C03637=1127.481,11.957,-50.735,179.626,6.543,149.306
C03638=1127.475,12.208,-50.749,179.627,6.548,149.306
C03639=1127.470,12.457,-50.763,179.628,6.553,149.307
C03640=1127.465,12.706,-50.777,179.629,6.558,149.308
C03641=1127.460,12.956,-50.790,179.630,6.562,149.309
C03642=1127.455,13.205,-50.804,179.630,6.567,149.309
C03643=1127.450,13.455,-50.818,179.632,6.572,149.310
C03644=1127.445,13.706,-50.832,179.632,6.576,149.311
C03645=1127.439,13.955,-50.846,179.633,6.581,149.312
C03646=1127.435,14.204,-50.860,179.634,6.585,149.312
C03647=1127.430,14.454,-50.874,179.635,6.590,149.313
C03648=1127.424,14.703,-50.887,179.636,6.594,149.314
C03649=1127.419,14.953,-50.901,179.637,6.600,149.315
C03650=1127.414,15.203,-50.916,179.638,6.604,149.315
C03651=1127.409,15.451,-50.929,179.639,6.609,149.316
C03652=1127.404,15.702,-50.942,179.640,6.613,149.317
C03653=1127.399,15.951,-50.957,179.640,6.618,149.318
C03654=1127.393,16.200,-50.971,179.642,6.622,149.318
C03655=1127.388,16.450,-50.985,179.643,6.627,149.319
C03656=1127.384,16.700,-50.999,179.644,6.632,149.320
C03657=1127.378,16.949,-51.013,179.645,6.636,149.321
C03658=1127.373,17.199,-51.027,179.646,6.640,149.321
C03659=1127.368,17.449,-51.040,179.646,6.645,149.322
C03660=1127.363,17.698,-51.054,179.647,6.649,149.323
C03661=1127.358,17.947,-51.069,179.649,6.655,149.323
C03662=1127.353,18.197,-51.083,179.650,6.659,149.324
C03663=1127.348,18.447,-51.097,179.651,6.664,149.325
C03664=1127.343,18.696,-51.111,179.652,6.668,149.326
C03665=1127.338,18.945,-51.125,179.652,6.673,149.326
C03666=1127.333,19.195,-51.140,179.653,6.677,149.327
C03667=1127.328,19.445,-51.154,179.654,6.681,149.328
C03668=1127.322,19.694,-51.168,179.656,6.686,149.328
C03669=1127.317,19.944,-51.182,179.657,6.691,149.329
C03670=1127.312,20.193,-51.196,179.658,6.695,149.330
C03671=1127.308,20.409,-51.208,179.658,6.699,149.331
C03672=1127.303,20.624,-51.220,179.659,6.703,149.331
C03673=1127.299,20.839,-51.233,179.661,6.707,149.332
C03674=1127.294,21.054,-51.245,179.661,6.711,149.332
C03675=1127.290,21.270,-51.257,179.662,6.715,149.333
C03676=1127.286,21.485,-51.270,179.662,6.719,149.334
C03677=1127.281,21.700,-51.281,179.664,6.723,149.334
C03678=1127.277,21.915,-51.294,179.664,6.726,149.335
C03679=1127.272,22.165,-51.309,179.665,6.730,149.335
C03680=1127.267,22.414,-51.323,179.667,6.736,149.336
C03681=1127.262,22.664,-51.337,179.668,6.740,149.337
C03682=1127.257,22.914,-51.351,179.669,6.745,149.337
C03683=1127.252,23.163,-51.366,179.670,6.749,149.338
C03684=1127.246,23.412,-51.380,179.671,6.753,149.339
C03685=1127.241,23.662,-51.394,179.672,6.758,149.339
C03686=1127.237,23.912,-51.408,179.673,6.762,149.340
C03687=1127.231,24.161,-51.424,179.674,6.767,149.341
C03688=1127.226,24.411,-51.438,179.675,6.771,149.342
C03689=1127.221,24.661,-51.452,179.676,6.776,149.342
C03690=1127.216,24.910,-51.466,179.677,6.780,149.343
C03691=1127.211,25.159,-51.480,179.678,6.785,149.344
C03692=1127.206,25.408,-51.495,179.679,6.789,149.344
C03693=1127.201,25.658,-51.510,179.680,6.793,149.345
C03694=1127.195,25.908,-51.525,179.682,6.798,149.345
C03695=1127.190,26.158,-51.539,179.683,6.802,149.346
C03696=1127.186,26.407,-51.554,179.684,6.806,149.347
C03697=1127.181,26.657,-51.568,179.684,6.811,149.348
C03698=1127.175,26.906,-51.582,179.685,6.815,149.348
C03699=1127.170,27.155,-51.596,179.686,6.820,149.349
C03700=1127.165,27.405,-51.612,179.688,6.825,149.350
C03701=1127.160,27.654,-51.626,179.689,6.829,149.350
C03702=1127.155,27.904,-51.640,179.690,6.833,149.351
C03703=1127.150,28.153,-51.655,179.691,6.838,149.352
C03704=1127.145,28.403,-51.670,179.692,6.842,149.352
C03705=1127.140,28.653,-51.685,179.693,6.846,149.353
C03706=1127.135,28.902,-51.700,179.694,6.851,149.353
C03707=1127.130,29.152,-51.714,179.695,6.855,149.354
C03708=1127.125,29.402,-51.728,179.696,6.859,149.355
C03709=1127.120,29.651,-51.744,179.697,6.863,149.355
C03710=1127.115,29.901,-51.758,179.699,6.868,149.356
C03711=1127.110,30.150,-51.773,179.700,6.872,149.357
C03712=1127.105,30.400,-51.788,179.701,6.876,149.357
C03713=1127.100,30.649,-51.802,179.702,6.881,149.358
C03714=1127.094,30.898,-51.817,179.703,6.886,149.359
C03715=1127.089,31.148,-51.832,179.704,6.890,149.359
C03716=1127.084,31.397,-51.847,179.706,6.894,149.360
C03717=1127.079,31.647,-51.861,179.707,6.898,149.360
C03718=1127.074,31.896,-51.876,179.708,6.903,149.361
C03719=1127.069,32.146,-51.891,179.709,6.907,149.362
C03720=1127.064,32.395,-51.906,179.710,6.911,149.362
C03721=1127.058,32.645,-51.921,179.711,6.916,149.363
C03722=1127.054,32.894,-51.936,179.712,6.920,149.364
C03723=1127.049,33.144,-51.950,179.713,6.924,149.364
C03724=1127.044,33.394,-51.966,179.714,6.929,149.365
C03725=1127.039,33.643,-51.981,179.716,6.933,149.366
C03726=1127.034,33.893,-51.995,179.717,6.937,149.366
C03727=1127.030,34.108,-52.008,179.718,6.941,149.367
C03728=1127.025,34.323,-52.021,179.719,6.944,149.367
C03729=1127.021,34.537,-52.034,179.720,6.949,149.368
C03730=1127.017,34.753,-52.047,179.721,6.952,149.368
C03731=1127.012,34.968,-52.060,179.722,6.956,149.369
C03732=1127.008,35.183,-52.073,179.723,6.959,149.369
C03733=1127.003,35.398,-52.085,179.724,6.963,149.370
C03734=1126.999,35.614,-52.099,179.725,6.967,149.370
C03735=1126.994,35.863,-52.114,179.726,6.971,149.371
C03736=1126.989,36.112,-52.129,179.727,6.975,149.372
C03737=1126.983,36.363,-52.144,179.728,6.980,149.372
C03738=1126.979,36.612,-52.159,179.730,6.983,149.373
C03739=1126.974,36.861,-52.174,179.731,6.988,149.373
C03740=1126.968,37.111,-52.189,179.732,6.992,149.374
C03741=1126.964,37.360,-52.204,179.733,6.996,149.375
C03742=1126.958,37.609,-52.219,179.734,7.001,149.375
C03743=1126.954,37.859,-52.235,179.736,7.005,149.376
C03744=1126.949,38.109,-52.250,179.737,7.009,149.376
C03745=1126.943,38.358,-52.265,179.738,7.013,149.377
C03746=1126.939,38.608,-52.280,179.739,7.018,149.378
C03747=1126.933,38.857,-52.296,179.740,7.021,149.378
C03748=1126.929,39.106,-52.311,179.741,7.026,149.379
C03749=1126.923,39.356,-52.326,179.742,7.030,149.379
C03750=1126.918,39.605,-52.341,179.744,7.034,149.380
C03751=1126.913,39.855,-52.357,179.745,7.038,149.380
C03752=1126.909,40.104,-52.372,179.746,7.043,149.381
C03753=1126.903,40.354,-52.387,179.747,7.047,149.382
C03754=1126.898,40.603,-52.403,179.748,7.051,149.382
C03755=1126.893,40.853,-52.417,179.750,7.055,149.383
C03756=1126.888,41.102,-52.433,179.751,7.059,149.383
C03757=1126.884,41.352,-52.448,179.752,7.064,149.384
C03758=1126.878,41.601,-52.464,179.753,7.068,149.384
C03759=1126.873,41.851,-52.479,179.755,7.072,149.385
C03760=1126.868,42.100,-52.494,179.756,7.076,149.386
C03761=1126.863,42.349,-52.510,179.757,7.080,149.386
C03762=1126.858,42.599,-52.526,179.758,7.085,149.387
C03763=1126.853,42.849,-52.541,179.759,7.089,149.387
C03764=1126.848,43.098,-52.556,179.761,7.093,149.388
C03765=1126.843,43.347,-52.572,179.762,7.097,149.389
C03766=1126.838,43.596,-52.587,179.763,7.101,149.389
C03767=1126.833,43.847,-52.603,179.765,7.105,149.390
C03768=1126.828,44.096,-52.618,179.766,7.110,149.390
C03769=1126.823,44.345,-52.633,179.767,7.114,149.391
C03770=1126.818,44.594,-52.649,179.768,7.118,149.391
C03771=1126.813,44.845,-52.665,179.769,7.122,149.392
C03772=1126.808,45.094,-52.681,179.770,7.126,149.393
C03773=1126.803,45.343,-52.696,179.772,7.130,149.393
C03774=1126.798,45.593,-52.711,179.773,7.135,149.394
C03775=1126.793,45.843,-52.727,179.775,7.139,149.394
C03776=1126.787,46.092,-52.743,179.776,7.143,149.395
C03777=1126.783,46.341,-52.758,179.777,7.147,149.395
C03778=1126.778,46.591,-52.774,179.778,7.151,149.396
C03779=1126.773,46.840,-52.790,179.779,7.155,149.396
C03780=1126.767,47.089,-52.805,179.781,7.159,149.397
C03781=1126.763,47.339,-52.821,179.782,7.164,149.398
C03782=1126.758,47.588,-52.836,179.783,7.168,149.398
C03783=1126.753,47.803,-52.849,179.785,7.172,149.399
C03784=1126.750,48.018,-52.864,179.786,7.175,149.399
C03785=1126.744,48.234,-52.877,179.787,7.179,149.399
C03786=1126.741,48.449,-52.891,179.788,7.182,149.400
C03787=1126.736,48.664,-52.904,179.789,7.186,149.401
C03788=1126.732,48.879,-52.918,179.790,7.189,149.401
C03789=1126.728,49.094,-52.931,179.791,7.193,149.401
C03790=1126.724,49.309,-52.945,179.793,7.197,149.402
C03791=1126.719,49.558,-52.961,179.794,7.201,149.402
C03792=1126.713,49.808,-52.976,179.795,7.205,149.403
C03793=1126.709,50.058,-52.992,179.796,7.209,149.404
C03794=1126.703,50.306,-53.009,179.798,7.213,149.404
C03795=1126.698,50.556,-53.024,179.799,7.217,149.405
C03796=1126.693,50.806,-53.040,179.801,7.221,149.405
C03797=1126.688,51.055,-53.057,179.802,7.225,149.406
C03798=1126.684,51.305,-53.072,179.803,7.229,149.406
C03799=1126.679,51.554,-53.088,179.804,7.234,149.407
C03800=1126.674,51.803,-53.104,179.806,7.238,149.407
C03801=1126.669,52.053,-53.120,179.807,7.242,149.408
C03802=1126.664,52.302,-53.135,179.808,7.246,149.408
C03803=1126.659,52.552,-53.152,179.810,7.250,149.409
C03804=1126.654,52.801,-53.168,179.811,7.254,149.409
C03805=1126.648,53.051,-53.183,179.812,7.258,149.410
C03806=1126.644,53.300,-53.200,179.813,7.261,149.410
C03807=1126.638,53.549,-53.215,179.814,7.266,149.411
C03808=1126.634,53.799,-53.232,179.816,7.270,149.411
C03809=1126.629,54.048,-53.248,179.817,7.274,149.412
C03810=1126.624,54.298,-53.264,179.818,7.278,149.413
C03811=1126.619,54.547,-53.280,179.820,7.282,149.413
C03812=1126.614,54.796,-53.296,179.821,7.286,149.414
C03813=1126.609,55.046,-53.312,179.822,7.290,149.414
C03814=1126.604,55.295,-53.329,179.824,7.294,149.415
C03815=1126.599,55.545,-53.345,179.825,7.298,149.415
C03816=1126.594,55.794,-53.361,179.826,7.303,149.416
C03817=1126.589,56.044,-53.377,179.828,7.306,149.416
C03818=1126.584,56.293,-53.393,179.829,7.311,149.417
C03819=1126.579,56.543,-53.409,179.831,7.315,149.417
C03820=1126.574,56.792,-53.425,179.832,7.319,149.418
C03821=1126.569,57.042,-53.442,179.833,7.323,149.418
C03822=1126.564,57.291,-53.458,179.835,7.327,149.419
C03823=1126.559,57.541,-53.474,179.836,7.331,149.419
C03824=1126.554,57.790,-53.490,179.837,7.335,149.420
C03825=1126.549,58.039,-53.507,179.839,7.339,149.420
C03826=1126.544,58.288,-53.523,179.840,7.343,149.421
C03827=1126.539,58.538,-53.539,179.841,7.347,149.422
C03828=1126.534,58.787,-53.556,179.843,7.351,149.422
C03829=1126.529,59.037,-53.572,179.844,7.355,149.422
C03830=1126.524,59.286,-53.589,179.845,7.360,149.423
C03831=1126.519,59.535,-53.605,179.847,7.363,149.423
C03832=1126.514,59.785,-53.621,179.849,7.367,149.424
C03833=1126.509,60.034,-53.637,179.850,7.372,149.425
C03834=1126.505,60.284,-53.654,179.851,7.376,149.425
C03835=1126.499,60.534,-53.670,179.852,7.379,149.426
C03836=1126.494,60.783,-53.687,179.853,7.383,149.426
C03837=1126.489,61.032,-53.703,179.855,7.387,149.426
C03838=1126.485,61.281,-53.720,179.856,7.391,149.427
C03839=1126.480,61.497,-53.735,179.858,7.395,149.428
C03840=1126.476,61.711,-53.748,179.858,7.398,149.428
C03841=1126.471,61.926,-53.763,179.860,7.402,149.428
C03842=1126.468,62.141,-53.777,179.861,7.405,149.429
C03843=1126.463,62.356,-53.791,179.862,7.408,149.429
C03844=1126.459,62.571,-53.805,179.863,7.412,149.430
C03845=1126.455,62.786,-53.820,179.864,7.415,149.430
C03846=1126.450,63.001,-53.834,179.866,7.419,149.431
C03847=1126.446,63.251,-53.850,179.868,7.423,149.431
C03848=1126.440,63.500,-53.867,179.869,7.428,149.432
C03849=1126.435,63.749,-53.883,179.870,7.431,149.432
C03850=1126.431,63.999,-53.900,179.872,7.435,149.432
C03851=1126.425,64.248,-53.917,179.872,7.439,149.433
C03852=1126.420,64.497,-53.934,179.874,7.443,149.434
C03853=1126.416,64.747,-53.950,179.875,7.447,149.434
C03854=1126.411,64.996,-53.967,179.877,7.451,149.435
C03855=1126.406,65.246,-53.984,179.878,7.455,149.435
C03856=1126.401,65.495,-54.000,179.880,7.459,149.435
C03857=1126.396,65.744,-54.016,179.881,7.463,149.436
C03858=1126.391,65.994,-54.033,179.882,7.467,149.437
C03859=1126.386,66.244,-54.050,179.884,7.471,149.437
C03860=1126.381,66.492,-54.066,179.885,7.475,149.438
C03861=1126.376,66.742,-54.084,179.887,7.479,149.438
C03862=1126.371,66.992,-54.100,179.888,7.483,149.438
C03863=1126.366,67.242,-54.117,179.890,7.487,149.439
C03864=1126.361,67.490,-54.134,179.891,7.491,149.440
C03865=1126.357,67.740,-54.150,179.892,7.495,149.440
C03866=1126.352,67.989,-54.168,179.894,7.499,149.440
C03867=1126.347,68.238,-54.185,179.895,7.503,149.441
C03868=1126.341,68.488,-54.202,179.897,7.507,149.441
C03869=1126.337,68.737,-54.219,179.898,7.511,149.442
C03870=1126.332,68.987,-54.235,179.900,7.515,149.442
C03871=1126.327,69.236,-54.252,179.901,7.519,149.443
C03872=1126.322,69.485,-54.269,179.903,7.523,149.443
C03873=1126.317,69.735,-54.286,179.904,7.527,149.444
C03874=1126.312,69.984,-54.303,179.905,7.531,149.444
C03875=1126.307,70.233,-54.320,179.907,7.535,149.445
C03876=1126.302,70.482,-54.337,179.908,7.538,149.445
C03877=1126.297,70.732,-54.354,179.909,7.542,149.446
C03878=1126.293,70.982,-54.371,179.910,7.547,149.446
C03879=1126.287,71.231,-54.388,179.912,7.551,149.447
C03880=1126.282,71.480,-54.405,179.914,7.554,149.447
C03881=1126.277,71.729,-54.423,179.915,7.558,149.448
C03882=1126.273,71.979,-54.439,179.916,7.563,149.448
C03883=1126.268,72.229,-54.457,179.918,7.567,149.449
C03884=1126.263,72.477,-54.473,179.919,7.570,149.449
C03885=1126.258,72.727,-54.491,179.921,7.574,149.450
C03886=1126.253,72.976,-54.508,179.922,7.579,149.450
C03887=1126.248,73.226,-54.525,179.924,7.583,149.451
C03888=1126.243,73.476,-54.542,179.925,7.586,149.451
C03889=1126.239,73.725,-54.559,179.926,7.591,149.452
C03890=1126.233,73.974,-54.576,179.928,7.595,149.452
C03891=1126.228,74.223,-54.594,179.930,7.599,149.453
C03892=1126.224,74.472,-54.611,179.931,7.602,149.453
C03893=1126.218,74.722,-54.628,179.933,7.606,149.453
C03894=1126.214,74.972,-54.645,179.934,7.611,149.454
C03895=1126.210,75.186,-54.660,179.935,7.614,149.455
C03896=1126.205,75.402,-54.675,179.936,7.618,149.455
C03897=1126.201,75.616,-54.690,179.937,7.621,149.455
C03898=1126.196,75.831,-54.705,179.939,7.624,149.456
C03899=1126.192,76.046,-54.720,179.940,7.627,149.456
C03900=1126.189,76.260,-54.735,179.941,7.630,149.456
C03901=1126.184,76.476,-54.749,179.943,7.634,149.457
C03902=1126.180,76.690,-54.765,179.944,7.637,149.457
C03903=1126.175,76.940,-54.782,179.945,7.642,149.458
C03904=1126.171,77.189,-54.800,179.946,7.645,149.458
C03905=1126.165,77.438,-54.816,179.947,7.649,149.459
C03906=1126.160,77.687,-54.834,179.948,7.652,149.459
C03907=1126.155,77.937,-54.852,179.948,7.656,149.460
C03908=1126.150,78.186,-54.868,179.950,7.660,149.461
C03909=1126.145,78.436,-54.886,179.951,7.663,149.461
C03910=1126.140,78.685,-54.904,179.952,7.667,149.462
C03911=1126.136,78.934,-54.921,179.953,7.671,149.462
C03912=1126.131,79.183,-54.939,179.954,7.675,149.463
C03913=1126.126,79.433,-54.956,179.955,7.678,149.463
C03914=1126.121,79.682,-54.974,179.956,7.682,149.464
C03915=1126.116,79.932,-54.991,179.957,7.685,149.464
C03916=1126.111,80.181,-55.009,179.958,7.690,149.465
C03917=1126.106,80.431,-55.026,179.960,7.694,149.465
C03918=1126.101,80.680,-55.044,179.960,7.697,149.466
C03919=1126.096,80.929,-55.062,179.962,7.701,149.466
C03920=1126.091,81.178,-55.078,179.962,7.704,149.467
C03921=1126.086,81.427,-55.096,179.964,7.708,149.468
C03922=1126.081,81.677,-55.114,179.965,7.713,149.468
C03923=1126.076,81.926,-55.132,179.966,7.716,149.469
C03924=1126.071,82.175,-55.150,179.967,7.720,149.469
C03925=1126.067,82.425,-55.166,179.968,7.723,149.470
C03926=1126.062,82.674,-55.184,179.969,7.727,149.470
C03927=1126.057,82.923,-55.202,179.971,7.731,149.471
C03928=1126.052,83.173,-55.219,179.972,7.734,149.471
C03929=1126.047,83.422,-55.237,179.973,7.739,149.472
C03930=1126.042,83.671,-55.255,179.974,7.743,149.472
C03931=1126.037,83.921,-55.273,179.975,7.746,149.473
C03932=1126.033,84.170,-55.290,179.976,7.750,149.473
C03933=1126.028,84.419,-55.308,179.978,7.754,149.474
C03934=1126.023,84.669,-55.326,179.979,7.758,149.474
C03935=1126.018,84.919,-55.344,179.980,7.761,149.475
C03936=1126.013,85.168,-55.362,179.982,7.765,149.475
C03937=1126.008,85.417,-55.380,179.983,7.770,149.476
C03938=1126.003,85.666,-55.398,179.984,7.773,149.476
C03939=1125.998,85.916,-55.415,179.985,7.777,149.477
C03940=1125.993,86.165,-55.433,179.987,7.781,149.477
C03941=1125.988,86.415,-55.451,179.988,7.785,149.478
C03942=1125.983,86.664,-55.469,179.990,7.789,149.478
C03943=1125.979,86.913,-55.486,179.991,7.793,149.479
C03944=1125.974,87.162,-55.504,179.992,7.796,149.479
C03945=1125.969,87.412,-55.521,179.993,7.800,149.480
C03946=1125.964,87.661,-55.539,179.995,7.804,149.480
C03947=1125.959,87.910,-55.557,179.996,7.808,149.481
C03948=1125.954,88.159,-55.575,179.998,7.812,149.481
C03949=1125.950,88.409,-55.594,179.999,7.816,149.482
C03950=1125.945,88.658,-55.612,-179.999,7.820,149.482
C03951=1125.941,88.873,-55.627,-179.998,7.823,149.483
C03952=1125.936,89.088,-55.643,-179.997,7.826,149.483
C03953=1125.932,89.303,-55.658,-179.996,7.830,149.483
C03954=1125.928,89.517,-55.674,-179.995,7.833,149.484
C03955=1125.924,89.732,-55.689,-179.994,7.836,149.484
C03956=1125.920,89.947,-55.705,-179.992,7.840,149.485
C03957=1125.916,90.162,-55.720,-179.991,7.843,149.485
C03958=1125.911,90.377,-55.736,-179.990,7.846,149.485
C03959=1125.906,90.626,-55.754,-179.988,7.850,149.486
C03960=1125.901,90.875,-55.772,-179.986,7.854,149.486
C03961=1125.896,91.124,-55.790,-179.985,7.858,149.487
C03962=1125.892,91.374,-55.808,-179.984,7.862,149.487
C03963=1125.887,91.623,-55.826,-179.982,7.866,149.488
C03964=1125.882,91.872,-55.844,-179.980,7.870,149.488
C03965=1125.877,92.121,-55.862,-179.979,7.873,149.489
C03966=1125.872,92.370,-55.881,-179.977,7.877,149.489
C03967=1125.867,92.619,-55.899,-179.976,7.881,149.489
C03968=1125.862,92.869,-55.918,-179.974,7.885,149.490
C03969=1125.857,93.119,-55.936,-179.973,7.889,149.490
C03970=1125.853,93.368,-55.954,-179.971,7.893,149.491
C03971=1125.848,93.617,-55.972,-179.969,7.898,149.491
C03972=1125.843,93.866,-55.990,-179.967,7.901,149.492
C03973=1125.838,94.116,-56.008,-179.965,7.905,149.492
C03974=1125.834,94.365,-56.027,-179.964,7.909,149.492
C03975=1125.828,94.614,-56.045,-179.962,7.913,149.493
C03976=1125.823,94.863,-56.063,-179.961,7.917,149.493
C03977=1125.819,95.113,-56.082,-179.959,7.921,149.493
C03978=1125.814,95.362,-56.100,-179.957,7.924,149.494
C03979=1125.809,95.611,-56.119,-179.955,7.928,149.494
C03980=1125.804,95.860,-56.137,-179.954,7.932,149.495
C03981=1125.799,96.110,-56.155,-179.952,7.936,149.495
C03982=1125.795,96.359,-56.173,-179.950,7.941,149.496
C03983=1125.790,96.608,-56.192,-179.948,7.945,149.496
C03984=1125.784,96.857,-56.211,-179.946,7.948,149.496
C03985=1125.780,97.107,-56.229,-179.945,7.952,149.497
C03986=1125.775,97.356,-56.248,-179.943,7.956,149.497
C03987=1125.770,97.605,-56.266,-179.942,7.960,149.498
C03988=1125.765,97.855,-56.284,-179.939,7.964,149.498
C03989=1125.761,98.104,-56.303,-179.937,7.968,149.498
C03990=1125.756,98.353,-56.321,-179.936,7.972,149.499
C03991=1125.751,98.603,-56.340,-179.934,7.976,149.499
C03992=1125.746,98.852,-56.359,-179.931,7.980,149.499
C03993=1125.741,99.101,-56.377,-179.930,7.984,149.500
C03994=1125.736,99.350,-56.395,-179.928,7.988,149.500
C03995=1125.732,99.600,-56.414,-179.926,7.991,149.500
C03996=1125.727,99.849,-56.432,-179.925,7.995,149.501
C03997=1125.722,100.098,-56.452,-179.922,8.000,149.501
C03998=1125.717,100.347,-56.470,-179.920,8.003,149.501
C03999=1125.712,100.596,-56.489,-179.919,8.007,149.502
C04000=1125.707,100.846,-56.508,-179.916,8.012,149.502
C04001=1125.703,101.095,-56.526,-179.914,8.015,149.502
C04002=1125.697,101.344,-56.545,-179.912,8.019,149.503
C04003=1125.693,101.594,-56.564,-179.911,8.023,149.503
C04004=1125.688,101.843,-56.583,-179.908,8.027,149.503
C04005=1125.683,102.092,-56.601,-179.906,8.031,149.504
C04006=1125.678,102.342,-56.620,-179.904,8.034,149.504
C04007=1125.674,102.556,-56.636,-179.903,8.038,149.504
C04008=1125.670,102.770,-56.653,-179.901,8.042,149.505
C04009=1125.666,102.986,-56.669,-179.899,8.045,149.505
C04010=1125.661,103.200,-56.685,-179.897,8.048,149.505
C04011=1125.657,103.415,-56.701,-179.896,8.052,149.506
C04012=1125.653,103.629,-56.718,-179.894,8.055,149.506
C04013=1125.650,103.844,-56.734,-179.891,8.059,149.506
C04014=1125.645,104.059,-56.750,-179.890,8.062,149.506
C04015=1125.640,104.308,-56.769,-179.888,8.066,149.507
C04016=1125.635,104.557,-56.788,-179.886,8.070,149.507
C04017=1125.630,104.806,-56.806,-179.883,8.074,149.507
C04018=1125.626,105.056,-56.826,-179.881,8.078,149.507
C04019=1125.621,105.305,-56.845,-179.879,8.082,149.508
C04020=1125.616,105.554,-56.864,-179.877,8.086,149.508
C04021=1125.611,105.804,-56.883,-179.875,8.089,149.508
C04022=1125.607,106.053,-56.902,-179.872,8.094,149.508
C04023=1125.601,106.302,-56.921,-179.870,8.098,149.509
C04024=1125.597,106.551,-56.940,-179.868,8.102,149.509
C04025=1125.592,106.800,-56.959,-179.866,8.105,149.509
C04026=1125.587,107.050,-56.979,-179.863,8.110,149.509
C04027=1125.582,107.299,-56.997,-179.861,8.113,149.510
C04028=1125.578,107.548,-57.017,-179.859,8.117,149.510
C04029=1125.573,107.797,-57.036,-179.857,8.121,149.510
C04030=1125.568,108.046,-57.055,-179.855,8.125,149.511
C04031=1125.563,108.295,-57.075,-179.852,8.129,149.511
C04032=1125.559,108.545,-57.093,-179.850,8.133,149.511
C04033=1125.553,108.794,-57.112,-179.847,8.137,149.511
C04034=1125.548,109.043,-57.132,-179.845,8.140,149.511
C04035=1125.544,109.293,-57.151,-179.842,8.145,149.512
C04036=1125.539,109.542,-57.170,-179.840,8.148,149.512
C04037=1125.534,109.791,-57.190,-179.838,8.152,149.512
C04038=1125.529,110.040,-57.209,-179.835,8.157,149.512
C04039=1125.525,110.289,-57.228,-179.833,8.160,149.513
C04040=1125.520,110.538,-57.247,-179.830,8.164,149.513
C04041=1125.515,110.788,-57.267,-179.828,8.168,149.513
C04042=1125.510,111.037,-57.287,-179.826,8.171,149.513
C04043=1125.506,111.286,-57.305,-179.824,8.175,149.513
C04044=1125.501,111.535,-57.325,-179.822,8.178,149.514
C04045=1125.496,111.784,-57.344,-179.820,8.182,149.514
C04046=1125.491,112.034,-57.364,-179.818,8.185,149.514
C04047=1125.486,112.283,-57.384,-179.816,8.189,149.514
C04048=1125.482,112.531,-57.403,-179.814,8.193,149.515
C04049=1125.477,112.781,-57.423,-179.812,8.196,149.515
C04050=1125.472,113.030,-57.442,-179.810,8.200,149.515
C04051=1125.467,113.279,-57.462,-179.808,8.204,149.516
C04052=1125.462,113.529,-57.481,-179.806,8.207,149.516
C04053=1125.457,113.779,-57.501,-179.804,8.211,149.516
C04054=1125.453,114.027,-57.520,-179.802,8.214,149.516
C04055=1125.448,114.276,-57.540,-179.801,8.217,149.516
C04056=1125.444,114.526,-57.560,-179.799,8.221,149.517
C04057=1125.438,114.774,-57.579,-179.797,8.224,149.517
C04058=1125.434,115.024,-57.599,-179.795,8.228,149.517
C04059=1125.429,115.274,-57.618,-179.793,8.231,149.518
C04060=1125.424,115.522,-57.638,-179.791,8.235,149.518
C04061=1125.419,115.771,-57.658,-179.789,8.239,149.518
C04062=1125.414,116.021,-57.678,-179.787,8.242,149.518
C04063=1125.410,116.235,-57.694,-179.786,8.245,149.519
C04064=1125.407,116.450,-57.712,-179.784,8.248,149.519
C04065=1125.402,116.664,-57.728,-179.782,8.251,149.519
C04066=1125.398,116.879,-57.745,-179.781,8.254,149.519
C04067=1125.394,117.094,-57.762,-179.779,8.257,149.520
C04068=1125.390,117.308,-57.780,-179.778,8.259,149.520
C04069=1125.385,117.522,-57.796,-179.776,8.263,149.520
C04070=1125.382,117.738,-57.814,-179.774,8.265,149.520
C04071=1125.377,117.986,-57.834,-179.772,8.269,149.520
C04072=1125.372,118.235,-57.853,-179.771,8.273,149.521
C04073=1125.367,118.485,-57.873,-179.769,8.276,149.521
C04074=1125.363,118.734,-57.893,-179.767,8.279,149.521
C04075=1125.358,118.983,-57.913,-179.765,8.283,149.522
C04076=1125.353,119.232,-57.933,-179.763,8.286,149.522
C04077=1125.348,119.481,-57.953,-179.762,8.290,149.522
C04078=1125.343,119.731,-57.972,-179.760,8.293,149.522
C04079=1125.339,119.980,-57.993,-179.758,8.296,149.523
C04080=1125.334,120.229,-58.012,-179.756,8.300,149.523
C04081=1125.329,120.478,-58.032,-179.754,8.303,149.523
C04082=1125.324,120.727,-58.052,-179.752,8.307,149.524
C04083=1125.320,120.976,-58.072,-179.751,8.310,149.524
C04084=1125.315,121.226,-58.092,-179.749,8.313,149.524
C04085=1125.310,121.475,-58.113,-179.747,8.317,149.524
C04086=1125.305,121.724,-58.132,-179.745,8.320,149.524
C04087=1125.300,121.973,-58.153,-179.744,8.323,149.525
C04088=1125.295,122.222,-58.172,-179.742,8.327,149.525
C04089=1125.291,122.471,-58.193,-179.740,8.330,149.525
C04090=1125.286,122.721,-58.212,-179.737,8.334,149.526
C04091=1125.282,122.970,-58.233,-179.736,8.337,149.526
C04092=1125.277,123.218,-58.253,-179.734,8.340,149.526
C04093=1125.272,123.468,-58.272,-179.732,8.344,149.526
C04094=1125.267,123.717,-58.293,-179.730,8.347,149.527
C04095=1125.262,123.966,-58.314,-179.729,8.350,149.527
C04096=1125.258,124.215,-58.333,-179.727,8.354,149.527
C04097=1125.253,124.464,-58.354,-179.725,8.357,149.527
C04098=1125.249,124.714,-58.373,-179.724,8.360,149.528
C04099=1125.243,124.963,-58.394,-179.722,8.364,149.528
C04100=1125.238,125.211,-58.414,-179.720,8.367,149.528
C04101=1125.234,125.460,-58.435,-179.718,8.371,149.529
C04102=1125.229,125.710,-58.454,-179.716,8.374,149.529
C04103=1125.225,125.959,-58.475,-179.714,8.377,149.529
C04104=1125.220,126.208,-58.496,-179.712,8.381,149.529
C04105=1125.215,126.458,-58.515,-179.711,8.384,149.530
C04106=1125.210,126.707,-58.536,-179.709,8.387,149.530
C04107=1125.206,126.956,-58.556,-179.707,8.391,149.530
C04108=1125.201,127.205,-58.577,-179.706,8.394,149.530
C04109=1125.196,127.454,-58.597,-179.704,8.397,149.531
C04110=1125.192,127.703,-58.617,-179.702,8.401,149.531
C04111=1125.187,127.952,-58.637,-179.701,8.404,149.531
C04112=1125.182,128.202,-58.658,-179.699,8.407,149.531
C04113=1125.178,128.451,-58.679,-179.697,8.411,149.532
C04114=1125.173,128.699,-58.699,-179.695,8.414,149.532
C04115=1125.167,128.949,-58.719,-179.693,8.417,149.532
C04116=1125.163,129.198,-58.739,-179.691,8.421,149.533
C04117=1125.158,129.447,-58.760,-179.690,8.424,149.533
C04118=1125.153,129.696,-58.781,-179.688,8.427,149.533
C04119=1125.149,129.910,-58.798,-179.687,8.430,149.533
C04120=1125.146,130.125,-58.816,-179.685,8.433,149.534
C04121=1125.141,130.339,-58.833,-179.684,8.435,149.534
C04122=1125.137,130.554,-58.851,-179.682,8.438,149.534
C04123=1125.133,130.769,-58.869,-179.681,8.441,149.535
C04124=1125.129,130.982,-58.887,-179.679,8.445,149.535
C04125=1125.125,131.197,-58.904,-179.678,8.447,149.535
C04126=1125.120,131.412,-58.922,-179.677,8.450,149.535
C04127=1125.116,131.661,-58.942,-179.675,8.453,149.535
C04128=1125.112,131.910,-58.963,-179.673,8.457,149.536
C04129=1125.106,132.159,-58.984,-179.671,8.460,149.536
C04130=1125.102,132.408,-59.004,-179.670,8.463,149.536
C04131=1125.097,132.658,-59.025,-179.668,8.466,149.537
C04132=1125.092,132.907,-59.045,-179.667,8.470,149.537
C04133=1125.087,133.156,-59.066,-179.665,8.473,149.537
C04134=1125.083,133.405,-59.087,-179.663,8.477,149.537
C04135=1125.078,133.653,-59.108,-179.662,8.480,149.538
C04136=1125.073,133.902,-59.129,-179.660,8.483,149.538
C04137=1125.069,134.151,-59.149,-179.659,8.486,149.539
C04138=1125.064,134.401,-59.170,-179.657,8.490,149.539
C04139=1125.059,134.650,-59.190,-179.654,8.493,149.539
C04140=1125.054,134.899,-59.211,-179.653,8.496,149.539
C04141=1125.050,135.148,-59.232,-179.651,8.500,149.540
C04142=1125.045,135.398,-59.253,-179.650,8.503,149.540
C04143=1125.041,135.647,-59.274,-179.648,8.506,149.540
C04144=1125.036,135.896,-59.294,-179.647,8.509,149.541
C04145=1125.031,136.144,-59.316,-179.645,8.513,149.541
C04146=1125.026,136.393,-59.337,-179.643,8.516,149.541
C04147=1125.021,136.643,-59.358,-179.642,8.519,149.541
C04148=1125.017,136.892,-59.378,-179.640,8.523,149.542
C04149=1125.011,137.141,-59.399,-179.639,8.526,149.542
C04150=1125.008,137.390,-59.420,-179.637,8.530,149.543
C04151=1125.003,137.639,-59.441,-179.636,8.532,149.543
C04152=1124.998,137.888,-59.462,-179.633,8.536,149.543
C04153=1124.993,138.137,-59.483,-179.632,8.539,149.543
C04154=1124.988,138.387,-59.504,-179.630,8.542,149.544
C04155=1124.984,138.635,-59.525,-179.629,8.546,149.544
C04156=1124.979,138.884,-59.546,-179.627,8.549,149.544
C04157=1124.975,139.134,-59.566,-179.626,8.553,149.545
C04158=1124.970,139.383,-59.588,-179.624,8.556,149.545
C04159=1124.965,139.632,-59.609,-179.623,8.559,149.545
C04160=1124.960,139.881,-59.629,-179.621,8.562,149.546
C04161=1124.955,140.130,-59.650,-179.620,8.566,149.546
C04162=1124.951,140.378,-59.671,-179.618,8.569,149.546
C04163=1124.946,140.628,-59.693,-179.616,8.573,149.547
C04164=1124.942,140.877,-59.714,-179.615,8.575,149.547
C04165=1124.937,141.126,-59.735,-179.613,8.579,149.547
C04166=1124.932,141.375,-59.756,-179.612,8.582,149.548
C04167=1124.927,141.624,-59.777,-179.610,8.586,149.548
C04168=1124.923,141.874,-59.798,-179.609,8.588,149.548
C04169=1124.918,142.123,-59.819,-179.607,8.592,149.549
C04170=1124.913,142.371,-59.841,-179.606,8.595,149.549
C04171=1124.909,142.620,-59.861,-179.604,8.599,149.549
C04172=1124.904,142.869,-59.883,-179.603,8.602,149.550
C04173=1124.899,143.119,-59.904,-179.601,8.606,149.550
C04174=1124.895,143.368,-59.926,-179.600,8.609,149.550
C04175=1124.891,143.582,-59.944,-179.599,8.611,149.551
C04176=1124.886,143.797,-59.962,-179.598,8.614,149.551
C04177=1124.883,144.011,-59.981,-179.596,8.617,149.551
C04178=1124.878,144.225,-59.999,-179.595,8.620,149.552
C04179=1124.874,144.439,-60.016,-179.594,8.623,149.552
C04180=1124.870,144.654,-60.035,-179.592,8.626,149.552
C04181=1124.866,144.868,-60.054,-179.591,8.629,149.553
C04182=1124.862,145.083,-60.072,-179.590,8.631,149.553
C04183=1124.857,145.332,-60.093,-179.587,8.636,149.553
C04184=1124.852,145.581,-60.114,-179.584,8.640,149.553
C04185=1124.848,145.830,-60.136,-179.582,8.643,149.554
C04186=1124.844,146.078,-60.157,-179.579,8.647,149.554
C04187=1124.839,146.328,-60.178,-179.576,8.652,149.554
C04188=1124.834,146.577,-60.200,-179.574,8.655,149.554
C04189=1124.829,146.826,-60.221,-179.572,8.659,149.554
C04190=1124.824,147.075,-60.243,-179.569,8.663,149.555
C04191=1124.820,147.324,-60.265,-179.567,8.667,149.555
C04192=1124.816,147.573,-60.285,-179.564,8.670,149.555
C04193=1124.811,147.822,-60.307,-179.562,8.674,149.555
C04194=1124.806,148.071,-60.329,-179.559,8.679,149.555
C04195=1124.801,148.320,-60.350,-179.557,8.682,149.556
C04196=1124.797,148.569,-60.372,-179.554,8.686,149.556
C04197=1124.792,148.818,-60.394,-179.551,8.690,149.556
C04198=1124.787,149.067,-60.416,-179.549,8.694,149.556
C04199=1124.782,149.316,-60.437,-179.546,8.697,149.556
C04200=1124.778,149.566,-60.459,-179.544,8.701,149.556
C04201=1124.773,149.814,-60.480,-179.541,8.705,149.557
C04202=1124.768,150.063,-60.502,-179.538,8.709,149.557
C04203=1124.764,150.312,-60.524,-179.536,8.712,149.557
C04204=1124.759,150.562,-60.545,-179.534,8.716,149.557
C04205=1124.754,150.810,-60.567,-179.531,8.719,149.557
C04206=1124.750,151.060,-60.589,-179.529,8.723,149.557
C04207=1124.745,151.308,-60.610,-179.526,8.727,149.558
C04208=1124.740,151.558,-60.632,-179.524,8.730,149.558
C04209=1124.736,151.806,-60.654,-179.521,8.735,149.558
C04210=1124.731,152.056,-60.676,-179.519,8.738,149.558
C04211=1124.726,152.304,-60.698,-179.516,8.741,149.558
C04212=1124.722,152.553,-60.720,-179.514,8.745,149.558
C04213=1124.717,152.802,-60.742,-179.511,8.749,149.558
C04214=1124.712,153.051,-60.763,-179.509,8.752,149.559
C04215=1124.708,153.301,-60.785,-179.506,8.756,149.559
C04216=1124.703,153.549,-60.806,-179.504,8.759,149.559
C04217=1124.699,153.798,-60.829,-179.501,8.763,149.559
C04218=1124.693,154.047,-60.851,-179.499,8.767,149.559
C04219=1124.689,154.296,-60.873,-179.496,8.770,149.559
C04220=1124.684,154.545,-60.895,-179.494,8.773,149.559
C04221=1124.680,154.794,-60.917,-179.491,8.777,149.559
C04222=1124.675,155.043,-60.939,-179.489,8.781,149.560
C04223=1124.671,155.292,-60.961,-179.486,8.784,149.560
C04224=1124.666,155.541,-60.983,-179.484,8.787,149.560
C04225=1124.661,155.791,-61.005,-179.481,8.791,149.560
C04226=1124.656,156.039,-61.027,-179.479,8.795,149.560
C04227=1124.652,156.289,-61.049,-179.476,8.798,149.560
C04228=1124.647,156.537,-61.071,-179.474,8.801,149.560
C04229=1124.643,156.786,-61.093,-179.472,8.804,149.560
C04230=1124.637,157.035,-61.116,-179.469,8.809,149.561
C04231=1124.633,157.249,-61.135,-179.467,8.811,149.561
C04232=1124.631,157.464,-61.154,-179.465,8.814,149.561
C04233=1124.627,157.678,-61.173,-179.463,8.817,149.561
C04234=1124.622,157.892,-61.192,-179.461,8.820,149.561
C04235=1124.618,158.106,-61.211,-179.458,8.823,149.561
C04236=1124.614,158.320,-61.230,-179.457,8.826,149.561
C04237=1124.610,158.535,-61.249,-179.454,8.829,149.561
C04238=1124.606,158.749,-61.268,-179.453,8.832,149.562
C04239=1124.601,158.998,-61.291,-179.450,8.835,149.562
C04240=1124.597,159.247,-61.313,-179.447,8.839,149.562
C04241=1124.592,159.496,-61.335,-179.445,8.842,149.562
C04242=1124.587,159.746,-61.358,-179.442,8.845,149.562
C04243=1124.583,159.994,-61.380,-179.440,8.848,149.562
C04244=1124.578,160.243,-61.402,-179.438,8.852,149.562
C04245=1124.573,160.493,-61.425,-179.435,8.855,149.562
C04246=1124.569,160.741,-61.447,-179.433,8.858,149.562
C04247=1124.565,160.990,-61.469,-179.431,8.861,149.562
C04248=1124.559,161.239,-61.492,-179.428,8.865,149.562
C04249=1124.555,161.488,-61.514,-179.426,8.868,149.563
C04250=1124.551,161.737,-61.536,-179.424,8.871,149.563
C04251=1124.546,161.985,-61.559,-179.420,8.875,149.563
C04252=1124.541,162.235,-61.581,-179.418,8.879,149.563
C04253=1124.537,162.484,-61.605,-179.416,8.882,149.563
C04254=1124.532,162.732,-61.627,-179.413,8.885,149.563
C04255=1124.528,162.981,-61.649,-179.411,8.888,149.563
C04256=1124.523,163.231,-61.672,-179.409,8.891,149.563
C04257=1124.519,163.479,-61.695,-179.406,8.894,149.563
C04258=1124.513,163.728,-61.717,-179.404,8.898,149.563
C04259=1124.509,163.977,-61.740,-179.402,8.901,149.564
C04260=1124.504,164.227,-61.762,-179.400,8.903,149.564
C04261=1124.500,164.475,-61.785,-179.397,8.907,149.564
C04262=1124.495,164.724,-61.808,-179.395,8.910,149.564
C04263=1124.491,164.973,-61.830,-179.393,8.913,149.564
C04264=1124.486,165.222,-61.854,-179.390,8.916,149.564
C04265=1124.481,165.471,-61.875,-179.388,8.920,149.564
C04266=1124.476,165.720,-61.899,-179.385,8.923,149.564
C04267=1124.472,165.968,-61.921,-179.383,8.926,149.564
C04268=1124.467,166.218,-61.944,-179.380,8.929,149.564
C04269=1124.463,166.466,-61.966,-179.378,8.932,149.565
C04270=1124.458,166.715,-61.990,-179.376,8.936,149.565
C04271=1124.454,166.965,-62.012,-179.373,8.939,149.565
C04272=1124.449,167.214,-62.035,-179.371,8.942,149.565
C04273=1124.445,167.462,-62.058,-179.369,8.945,149.565
C04274=1124.440,167.711,-62.081,-179.367,8.948,149.565
C04275=1124.435,167.960,-62.104,-179.364,8.951,149.565
C04276=1124.431,168.209,-62.126,-179.362,8.954,149.565
C04277=1124.426,168.457,-62.149,-179.360,8.957,149.565
C04278=1124.421,168.706,-62.173,-179.357,8.960,149.565
C04279=1124.417,168.955,-62.195,-179.355,8.964,149.565
C04280=1124.412,169.205,-62.218,-179.353,8.966,149.566
C04281=1124.408,169.453,-62.241,-179.351,8.969,149.566
C04282=1124.403,169.702,-62.264,-179.348,8.972,149.566
C04283=1124.398,169.951,-62.287,-179.346,8.976,149.566
C04284=1124.394,170.200,-62.310,-179.343,8.979,149.566
C04285=1124.389,170.449,-62.333,-179.341,8.981,149.566
C04286=1124.384,170.698,-62.356,-179.339,8.985,149.566
C04287=1124.381,170.912,-62.376,-179.338,8.987,149.566
C04288=1124.376,171.126,-62.396,-179.335,8.990,149.566
C04289=1124.373,171.341,-62.416,-179.333,8.993,149.566
C04290=1124.369,171.554,-62.435,-179.331,8.995,149.566
C04291=1124.365,171.769,-62.455,-179.330,8.998,149.567
C04292=1124.361,171.983,-62.475,-179.327,9.001,149.567
C04293=1124.357,172.196,-62.495,-179.325,9.003,149.567
C04294=1124.353,172.412,-62.515,-179.323,9.005,149.567
C04295=1124.348,172.660,-62.538,-179.321,9.009,149.567
C04296=1124.344,172.909,-62.561,-179.319,9.012,149.567
C04297=1124.339,173.158,-62.584,-179.317,9.014,149.567
C04298=1124.334,173.407,-62.608,-179.314,9.017,149.567
C04299=1124.329,173.656,-62.631,-179.312,9.021,149.567
C04300=1124.325,173.905,-62.654,-179.310,9.023,149.567
C04301=1124.321,174.153,-62.678,-179.308,9.026,149.567
C04302=1124.316,174.402,-62.701,-179.306,9.030,149.568
C04303=1124.312,174.651,-62.724,-179.303,9.033,149.568
C04304=1124.307,174.900,-62.748,-179.301,9.035,149.568
C04305=1124.303,175.149,-62.771,-179.299,9.038,149.568
C04306=1124.298,175.398,-62.794,-179.297,9.042,149.568
C04307=1124.293,175.646,-62.817,-179.295,9.044,149.568
C04308=1124.288,175.895,-62.840,-179.292,9.047,149.568
C04309=1124.284,176.144,-62.864,-179.290,9.051,149.568
C04310=1124.279,176.393,-62.888,-179.288,9.053,149.568
C04311=1124.275,176.641,-62.911,-179.286,9.056,149.568
C04312=1124.271,176.890,-62.934,-179.284,9.060,149.568
C04313=1124.266,177.139,-62.957,-179.282,9.062,149.569
C04314=1124.261,177.388,-62.981,-179.279,9.065,149.569
C04315=1124.257,177.637,-63.005,-179.278,9.068,149.569
C04316=1124.252,177.886,-63.028,-179.275,9.071,149.569
C04317=1124.247,178.135,-63.051,-179.273,9.074,149.569
C04318=1124.243,178.384,-63.075,-179.271,9.077,149.569
C04319=1124.238,178.632,-63.099,-179.269,9.080,149.569
C04320=1124.234,178.881,-63.122,-179.266,9.083,149.569
C04321=1124.229,179.130,-63.146,-179.265,9.086,149.569
C04322=1124.225,179.379,-63.168,-179.262,9.089,149.569
C04323=1124.221,179.628,-63.192,-179.259,9.093,149.569
C04324=1124.216,179.877,-63.216,-179.256,9.095,149.569
C04325=1124.211,180.126,-63.239,-179.254,9.099,149.569
C04326=1124.207,180.374,-63.263,-179.251,9.102,149.569
C04327=1124.202,180.623,-63.287,-179.248,9.106,149.569
C04328=1124.198,180.873,-63.310,-179.245,9.109,149.570
C04329=1124.194,181.121,-63.334,-179.242,9.112,149.569
C04330=1124.189,181.370,-63.358,-179.239,9.115,149.569
C04331=1124.184,181.619,-63.382,-179.237,9.118,149.569
C04332=1124.180,181.868,-63.405,-179.234,9.122,149.569
C04333=1124.175,182.116,-63.430,-179.231,9.125,149.569
C04334=1124.170,182.365,-63.453,-179.228,9.128,149.569
C04335=1124.165,182.614,-63.477,-179.226,9.131,149.569
C04336=1124.161,182.863,-63.501,-179.223,9.134,149.569
C04337=1124.156,183.111,-63.525,-179.221,9.137,149.570
C04338=1124.152,183.360,-63.548,-179.218,9.140,149.569
C04339=1124.148,183.609,-63.572,-179.215,9.143,149.569
C04340=1124.143,183.858,-63.596,-179.213,9.146,149.569
C04341=1124.139,184.107,-63.620,-179.210,9.150,149.569
C04342=1124.134,184.356,-63.643,-179.208,9.153,149.570
C04343=1124.130,184.569,-63.664,-179.205,9.155,149.569
C04344=1124.126,184.784,-63.685,-179.203,9.158,149.569
C04345=1124.122,184.998,-63.706,-179.200,9.161,149.569
C04346=1124.118,185.212,-63.726,-179.198,9.163,149.569
C04347=1124.114,185.426,-63.746,-179.196,9.165,149.569
C04348=1124.110,185.640,-63.768,-179.194,9.169,149.570
C04349=1124.106,185.854,-63.788,-179.192,9.171,149.570
C04350=1124.102,186.068,-63.808,-179.190,9.173,149.570
C04351=1124.098,186.317,-63.833,-179.187,9.176,149.569
C04352=1124.094,186.566,-63.857,-179.185,9.179,149.569
C04353=1124.089,186.815,-63.881,-179.182,9.182,149.570
C04354=1124.084,187.063,-63.905,-179.180,9.185,149.570
C04355=1124.080,187.312,-63.929,-179.178,9.188,149.570
C04356=1124.075,187.562,-63.953,-179.175,9.191,149.570
C04357=1124.071,187.810,-63.977,-179.173,9.193,149.570
C04358=1124.066,188.058,-64.001,-179.171,9.196,149.570
C04359=1124.061,188.307,-64.026,-179.168,9.199,149.570
C04360=1124.057,188.556,-64.050,-179.166,9.202,149.570
C04361=1124.053,188.805,-64.074,-179.164,9.205,149.570
C04362=1124.048,189.054,-64.098,-179.162,9.207,149.570
C04363=1124.043,189.302,-64.122,-179.159,9.210,149.570
C04364=1124.039,189.551,-64.147,-179.157,9.212,149.570
C04365=1124.035,189.800,-64.171,-179.155,9.216,149.570
C04366=1124.030,190.049,-64.195,-179.153,9.218,149.570
C04367=1124.025,190.298,-64.219,-179.151,9.221,149.570
C04368=1124.021,190.546,-64.243,-179.149,9.223,149.570
C04369=1124.016,190.796,-64.268,-179.147,9.227,149.570
C04370=1124.012,191.044,-64.292,-179.145,9.229,149.570
C04371=1124.008,191.292,-64.316,-179.142,9.232,149.570
C04372=1124.002,191.541,-64.341,-179.140,9.235,149.571
C04373=1123.999,191.790,-64.365,-179.138,9.237,149.571
C04374=1123.994,192.039,-64.390,-179.136,9.240,149.571
C04375=1123.989,192.287,-64.414,-179.134,9.243,149.571
C04376=1123.985,192.536,-64.439,-179.132,9.245,149.571
C04377=1123.980,192.785,-64.463,-179.131,9.247,149.571
C04378=1123.976,193.034,-64.487,-179.128,9.251,149.571
C04379=1123.971,193.282,-64.512,-179.127,9.253,149.571
C04380=1123.967,193.531,-64.536,-179.125,9.256,149.571
C04381=1123.962,193.780,-64.561,-179.123,9.258,149.571
C04382=1123.957,194.029,-64.585,-179.121,9.261,149.572
C04383=1123.954,194.278,-64.610,-179.119,9.264,149.572
C04384=1123.948,194.526,-64.634,-179.117,9.266,149.572
C04385=1123.944,194.775,-64.658,-179.116,9.269,149.572
C04386=1123.939,195.024,-64.683,-179.114,9.271,149.572
C04387=1123.935,195.273,-64.707,-179.113,9.274,149.572
C04388=1123.930,195.521,-64.732,-179.111,9.276,149.572
C04389=1123.926,195.771,-64.757,-179.109,9.279,149.573
C04390=1123.921,196.019,-64.781,-179.107,9.281,149.573
C04391=1123.917,196.268,-64.805,-179.106,9.284,149.573
C04392=1123.912,196.517,-64.830,-179.103,9.288,149.573
C04393=1123.908,196.765,-64.855,-179.099,9.292,149.573
C04394=1123.903,197.014,-64.880,-179.095,9.295,149.573
C04395=1123.899,197.263,-64.904,-179.092,9.299,149.572
C04396=1123.894,197.511,-64.929,-179.089,9.302,149.573
C04397=1123.890,197.761,-64.953,-179.085,9.306,149.572
C04398=1123.885,198.009,-64.979,-179.082,9.310,149.572
C04399=1123.881,198.223,-64.999,-179.078,9.313,149.572
C04400=1123.878,198.437,-65.021,-179.075,9.316,149.572
C04401=1123.874,198.650,-65.042,-179.072,9.319,149.572
C04402=1123.870,198.864,-65.064,-179.070,9.322,149.572
C04403=1123.866,199.078,-65.085,-179.067,9.324,149.572
C04404=1123.862,199.293,-65.106,-179.064,9.327,149.572
C04405=1123.858,199.507,-65.128,-179.061,9.330,149.572
C04406=1123.854,199.720,-65.149,-179.058,9.333,149.571
C04407=1123.850,199.969,-65.174,-179.055,9.336,149.571
C04408=1123.845,200.218,-65.199,-179.051,9.340,149.571
C04409=1123.841,200.467,-65.224,-179.048,9.343,149.571
C04410=1123.837,200.715,-65.249,-179.044,9.346,149.571
C04411=1123.832,200.964,-65.274,-179.042,9.349,149.571
C04412=1123.827,201.212,-65.299,-179.038,9.353,149.571
C04413=1123.824,201.462,-65.323,-179.035,9.356,149.571
C04414=1123.818,201.710,-65.348,-179.032,9.359,149.571
C04415=1123.814,201.959,-65.374,-179.029,9.362,149.570
C04416=1123.809,202.208,-65.399,-179.025,9.365,149.570
C04417=1123.806,202.456,-65.424,-179.022,9.368,149.570
C04418=1123.800,202.705,-65.448,-179.019,9.371,149.570
C04419=1123.796,202.954,-65.474,-179.016,9.375,149.570
C04420=1123.791,203.202,-65.500,-179.013,9.377,149.570
C04421=1123.788,203.451,-65.524,-179.010,9.380,149.570
C04422=1123.783,203.700,-65.550,-179.007,9.383,149.570
C04423=1123.778,203.949,-65.574,-179.004,9.386,149.569
C04424=1123.774,204.197,-65.600,-179.001,9.389,149.569
C04425=1123.769,204.445,-65.626,-178.998,9.392,149.569
C04426=1123.765,204.695,-65.651,-178.995,9.395,149.569
C04427=1123.761,204.943,-65.675,-178.992,9.398,149.569
C04428=1123.756,205.192,-65.700,-178.989,9.401,149.569
C04429=1123.752,205.441,-65.726,-178.987,9.404,149.569
C04430=1123.747,205.689,-65.752,-178.984,9.406,149.569
C04431=1123.743,205.938,-65.777,-178.981,9.409,149.569
C04432=1123.738,206.187,-65.802,-178.978,9.412,149.569
C04433=1123.733,206.435,-65.828,-178.976,9.415,149.569
C04434=1123.729,206.684,-65.853,-178.973,9.418,149.568
C04435=1123.724,206.932,-65.879,-178.970,9.421,149.569
C04436=1123.720,207.182,-65.904,-178.967,9.424,149.568
C04437=1123.716,207.429,-65.929,-178.965,9.426,149.568
C04438=1123.712,207.678,-65.954,-178.962,9.429,149.568
C04439=1123.707,207.927,-65.980,-178.960,9.432,149.568
C04440=1123.702,208.176,-66.005,-178.957,9.435,149.568
C04441=1123.698,208.425,-66.031,-178.955,9.437,149.568
C04442=1123.694,208.673,-66.056,-178.952,9.440,149.568
C04443=1123.689,208.922,-66.082,-178.949,9.443,149.568
C04444=1123.685,209.170,-66.107,-178.947,9.446,149.568
C04445=1123.680,209.419,-66.133,-178.945,9.448,149.568
C04446=1123.676,209.667,-66.159,-178.942,9.451,149.568
C04447=1123.671,209.916,-66.184,-178.940,9.454,149.568
C04448=1123.667,210.165,-66.210,-178.938,9.456,149.568
C04449=1123.662,210.414,-66.235,-178.935,9.459,149.568
C04450=1123.658,210.662,-66.261,-178.933,9.461,149.568
C04451=1123.653,210.911,-66.287,-178.930,9.465,149.568
C04452=1123.649,211.160,-66.313,-178.928,9.467,149.568
C04453=1123.644,211.408,-66.338,-178.926,9.470,149.568
C04454=1123.640,211.657,-66.364,-178.924,9.472,149.568
C04455=1123.636,211.871,-66.386,-178.922,9.475,149.568
C04456=1123.632,212.085,-66.408,-178.920,9.477,149.568
C04457=1123.629,212.298,-66.430,-178.918,9.479,149.568
C04458=1123.624,212.512,-66.452,-178.917,9.482,149.569
C04459=1123.621,212.726,-66.474,-178.915,9.484,149.569
C04460=1123.617,212.940,-66.497,-178.913,9.487,149.569
C04461=1123.613,213.153,-66.519,-178.911,9.489,149.569
C04462=1123.609,213.368,-66.541,-178.910,9.492,149.569
C04463=1123.605,213.616,-66.567,-178.908,9.494,149.569
C04464=1123.601,213.865,-66.592,-178.906,9.496,149.569
C04465=1123.596,214.113,-66.618,-178.904,9.500,149.569
C04466=1123.592,214.362,-66.644,-178.902,9.502,149.569
C04467=1123.588,214.610,-66.670,-178.900,9.506,149.570
C04468=1123.583,214.859,-66.696,-178.898,9.508,149.570
C04469=1123.578,215.108,-66.722,-178.896,9.510,149.570
C04470=1123.574,215.356,-66.747,-178.894,9.514,149.570
C04471=1123.569,215.605,-66.773,-178.892,9.516,149.570
C04472=1123.565,215.853,-66.800,-178.890,9.520,149.570
C04473=1123.561,216.102,-66.825,-178.888,9.522,149.570
C04474=1123.556,216.351,-66.852,-178.885,9.525,149.571
C04475=1123.551,216.599,-66.877,-178.883,9.528,149.571
C04476=1123.547,216.848,-66.903,-178.881,9.531,149.571
C04477=1123.543,217.096,-66.929,-178.879,9.534,149.571
C04478=1123.538,217.345,-66.956,-178.877,9.537,149.571
C04479=1123.534,217.594,-66.981,-178.875,9.540,149.571
C04480=1123.529,217.842,-67.007,-178.872,9.543,149.571
C04481=1123.525,218.091,-67.033,-178.870,9.546,149.571
C04482=1123.520,218.340,-67.060,-178.868,9.549,149.572
C04483=1123.516,218.588,-67.085,-178.866,9.552,149.572
C04484=1123.512,218.837,-67.112,-178.863,9.555,149.572
C04485=1123.508,219.085,-67.138,-178.861,9.558,149.572
C04486=1123.503,219.335,-67.164,-178.858,9.561,149.572
C04487=1123.499,219.583,-67.190,-178.856,9.565,149.572
C04488=1123.494,219.831,-67.216,-178.854,9.568,149.572
C04489=1123.489,220.080,-67.242,-178.851,9.571,149.572
C04490=1123.485,220.328,-67.269,-178.849,9.574,149.572
C04491=1123.481,220.577,-67.294,-178.846,9.577,149.572
C04492=1123.476,220.825,-67.321,-178.844,9.580,149.572
C04493=1123.472,221.074,-67.347,-178.841,9.583,149.572
C04494=1123.468,221.323,-67.373,-178.838,9.586,149.573
C04495=1123.463,221.572,-67.400,-178.836,9.589,149.573
C04496=1123.459,221.820,-67.426,-178.833,9.593,149.573
C04497=1123.455,222.069,-67.453,-178.831,9.596,149.573
C04498=1123.450,222.317,-67.478,-178.828,9.599,149.573
C04499=1123.446,222.565,-67.505,-178.826,9.602,149.573
C04500=1123.441,222.814,-67.531,-178.823,9.606,149.573
C04501=1123.437,223.062,-67.557,-178.820,9.609,149.573
C04502=1123.432,223.311,-67.585,-178.817,9.612,149.573
C04503=1123.428,223.560,-67.610,-178.815,9.615,149.573
C04504=1123.423,223.808,-67.637,-178.812,9.619,149.573
C04505=1123.419,224.057,-67.663,-178.809,9.622,149.573
C04506=1123.414,224.306,-67.690,-178.806,9.625,149.573
C04507=1123.411,224.554,-67.717,-178.804,9.628,149.573
C04508=1123.406,224.803,-67.742,-178.800,9.631,149.573
C04509=1123.402,225.051,-67.769,-178.798,9.635,149.573
C04510=1123.397,225.300,-67.796,-178.794,9.638,149.573
C04511=1123.394,225.513,-67.819,-178.792,9.640,149.573
C04512=1123.390,225.727,-67.841,-178.789,9.643,149.573
C04513=1123.386,225.941,-67.865,-178.787,9.646,149.573
C04514=1123.382,226.155,-67.887,-178.784,9.649,149.573
C04515=1123.378,226.368,-67.910,-178.781,9.652,149.573
C04516=1123.374,226.582,-67.933,-178.779,9.655,149.573
C04517=1123.371,226.796,-67.956,-178.777,9.657,149.573
C04518=1123.367,227.010,-67.979,-178.774,9.660,149.573
C04519=1123.363,227.258,-68.005,-178.770,9.664,149.573
C04520=1123.358,227.507,-68.032,-178.768,9.667,149.573
C04521=1123.354,227.755,-68.059,-178.764,9.670,149.573
C04522=1123.349,228.003,-68.086,-178.761,9.674,149.573
C04523=1123.345,228.252,-68.113,-178.758,9.677,149.573
C04524=1123.341,228.500,-68.139,-178.754,9.680,149.572
C04525=1123.336,228.749,-68.166,-178.751,9.684,149.572
C04526=1123.331,228.997,-68.193,-178.748,9.687,149.572
C04527=1123.327,229.246,-68.219,-178.745,9.690,149.572
C04528=1123.323,229.495,-68.247,-178.741,9.694,149.572
C04529=1123.319,229.743,-68.274,-178.738,9.697,149.572
C04530=1123.315,229.992,-68.300,-178.734,9.700,149.572
C04531=1123.310,230.240,-68.327,-178.731,9.704,149.572
C04532=1123.305,230.489,-68.354,-178.727,9.706,149.571
C04533=1123.301,230.737,-68.381,-178.724,9.710,149.571
C04534=1123.297,230.985,-68.408,-178.720,9.713,149.571
C04535=1123.292,231.234,-68.435,-178.717,9.716,149.571
C04536=1123.288,231.483,-68.462,-178.714,9.719,149.571
C04537=1123.283,231.731,-68.490,-178.711,9.722,149.571
C04538=1123.280,231.980,-68.516,-178.708,9.725,149.571
C04539=1123.275,232.228,-68.543,-178.704,9.728,149.571
C04540=1123.270,232.477,-68.570,-178.701,9.731,149.570
C04541=1123.266,232.725,-68.598,-178.698,9.734,149.570
C04542=1123.262,232.974,-68.625,-178.695,9.737,149.570
C04543=1123.258,233.222,-68.652,-178.692,9.740,149.570
C04544=1123.253,233.470,-68.679,-178.689,9.743,149.570
C04545=1123.249,233.719,-68.706,-178.686,9.746,149.570
C04546=1123.245,233.968,-68.733,-178.683,9.748,149.570
C04547=1123.240,234.216,-68.761,-178.679,9.752,149.570
C04548=1123.236,234.464,-68.788,-178.677,9.755,149.570
C04549=1123.231,234.713,-68.815,-178.674,9.757,149.569
C04550=1123.227,234.961,-68.842,-178.671,9.760,149.569
C04551=1123.223,235.210,-68.870,-178.668,9.763,149.569
C04552=1123.219,235.458,-68.897,-178.665,9.766,149.569
C04553=1123.214,235.707,-68.924,-178.662,9.769,149.569
C04554=1123.210,235.955,-68.952,-178.659,9.772,149.569
C04555=1123.205,236.204,-68.979,-178.657,9.774,149.569
C04556=1123.201,236.452,-69.006,-178.654,9.776,149.569
C04557=1123.196,236.700,-69.034,-178.651,9.779,149.569
C04558=1123.192,236.949,-69.061,-178.648,9.782,149.568
C04559=1123.188,237.198,-69.089,-178.645,9.785,149.568
C04560=1123.183,237.446,-69.116,-178.643,9.787,149.568
C04561=1123.179,237.694,-69.143,-178.640,9.790,149.568
C04562=1123.175,237.943,-69.171,-178.637,9.792,149.568
C04563=1123.170,238.191,-69.199,-178.635,9.794,149.568
C04564=1123.166,238.439,-69.226,-178.633,9.797,149.568
C04565=1123.162,238.688,-69.254,-178.630,9.799,149.568
C04566=1123.157,238.937,-69.281,-178.627,9.802,149.568
C04567=1123.154,239.151,-69.305,-178.625,9.804,149.568
C04568=1123.150,239.364,-69.329,-178.623,9.806,149.568
C04569=1123.146,239.577,-69.352,-178.621,9.809,149.568
C04570=1123.143,239.791,-69.376,-178.619,9.811,149.568
C04571=1123.139,240.004,-69.399,-178.617,9.813,149.568
C04572=1123.135,240.218,-69.423,-178.615,9.815,149.568
C04573=1123.131,240.431,-69.447,-178.613,9.817,149.568
C04574=1123.128,240.645,-69.471,-178.610,9.819,149.567
C04575=1123.124,240.893,-69.499,-178.609,9.822,149.568
C04576=1123.119,241.142,-69.527,-178.606,9.824,149.567
C04577=1123.115,241.390,-69.554,-178.604,9.827,149.567
C04578=1123.110,241.639,-69.581,-178.601,9.829,149.567
C04579=1123.106,241.887,-69.610,-178.600,9.831,149.567
C04580=1123.101,242.136,-69.637,-178.598,9.833,149.567
C04581=1123.097,242.384,-69.664,-178.595,9.836,149.567
C04582=1123.093,242.632,-69.693,-178.593,9.838,149.567
C04583=1123.089,242.881,-69.720,-178.591,9.841,149.567
C04584=1123.084,243.130,-69.748,-178.589,9.843,149.567
C04585=1123.080,243.378,-69.776,-178.587,9.845,149.567
C04586=1123.075,243.626,-69.803,-178.585,9.847,149.567
C04587=1123.071,243.875,-69.831,-178.583,9.850,149.567
C04588=1123.067,244.123,-69.859,-178.581,9.852,149.568
C04589=1123.063,244.371,-69.887,-178.579,9.854,149.568
C04590=1123.058,244.620,-69.915,-178.577,9.857,149.568
C04591=1123.054,244.868,-69.943,-178.575,9.859,149.568
C04592=1123.050,245.116,-69.971,-178.573,9.861,149.568
C04593=1123.045,245.365,-69.998,-178.572,9.864,149.568
C04594=1123.041,245.614,-70.027,-178.570,9.866,149.568
C04595=1123.036,245.862,-70.054,-178.568,9.869,149.568
C04596=1123.033,246.110,-70.083,-178.566,9.871,149.568
C04597=1123.028,246.358,-70.110,-178.564,9.873,149.568
C04598=1123.024,246.607,-70.138,-178.563,9.876,149.569
C04599=1123.019,246.855,-70.166,-178.562,9.878,149.569
C04600=1123.015,247.104,-70.194,-178.560,9.880,149.569
C04601=1123.011,247.352,-70.222,-178.558,9.883,149.569
C04602=1123.006,247.600,-70.250,-178.555,9.886,149.569
C04603=1123.002,247.849,-70.279,-178.548,9.891,149.568
C04604=1122.998,248.097,-70.306,-178.543,9.896,149.568
C04605=1122.994,248.346,-70.334,-178.537,9.900,149.567
C04606=1122.989,248.594,-70.362,-178.532,9.905,149.567
C04607=1122.985,248.843,-70.390,-178.526,9.909,149.567
C04608=1122.980,249.091,-70.419,-178.521,9.913,149.566
C04609=1122.976,249.339,-70.447,-178.516,9.917,149.566
C04610=1122.972,249.588,-70.475,-178.512,9.921,149.566
C04611=1122.967,249.836,-70.503,-178.507,9.924,149.565
C04612=1122.964,250.085,-70.531,-178.502,9.928,149.565
C04613=1122.958,250.333,-70.560,-178.498,9.931,149.565
C04614=1122.955,250.581,-70.589,-178.494,9.935,149.564
C04615=1122.951,250.829,-70.616,-178.490,9.938,149.564
C04616=1122.946,251.078,-70.645,-178.486,9.941,149.564
C04617=1122.942,251.326,-70.673,-178.483,9.943,149.563
C04618=1122.937,251.574,-70.702,-178.479,9.947,149.563
C04619=1122.934,251.823,-70.730,-178.476,9.949,149.563
C04620=1122.929,252.070,-70.759,-178.473,9.952,149.563
C04621=1122.925,252.319,-70.787,-178.470,9.954,149.563
C04622=1122.921,252.568,-70.816,-178.467,9.956,149.563
C04623=1122.916,252.781,-70.840,-178.465,9.958,149.562
C04624=1122.913,252.994,-70.865,-178.464,9.960,149.562
C04625=1122.909,253.208,-70.889,-178.461,9.962,149.562
C04626=1122.906,253.422,-70.914,-178.459,9.964,149.562
C04627=1122.902,253.635,-70.938,-178.458,9.965,149.562
C04628=1122.899,253.848,-70.963,-178.457,9.967,149.562
C04629=1122.895,254.062,-70.987,-178.455,9.969,149.562
C04630=1122.891,254.275,-71.012,-178.454,9.970,149.562
C04631=1122.887,254.524,-71.040,-178.453,9.972,149.562
C04632=1122.882,254.772,-71.069,-178.451,9.973,149.562
C04633=1122.878,255.020,-71.098,-178.450,9.975,149.562
C04634=1122.874,255.269,-71.126,-178.450,9.976,149.563
C04635=1122.870,255.517,-71.154,-178.450,9.977,149.563
C04636=1122.865,255.765,-71.183,-178.449,9.979,149.563
C04637=1122.861,256.014,-71.212,-178.449,9.980,149.563
C04638=1122.857,256.262,-71.240,-178.446,9.983,149.563
C04639=1122.852,256.510,-71.269,-178.443,9.986,149.563
C04640=1122.848,256.758,-71.298,-178.440,9.988,149.563
C04641=1122.844,257.007,-71.327,-178.437,9.991,149.563
C04642=1122.839,257.255,-71.355,-178.434,9.994,149.563
C04643=1122.835,257.503,-71.384,-178.431,9.997,149.563
C04644=1122.831,257.752,-71.413,-178.429,10.000,149.563
C04645=1122.826,258.000,-71.441,-178.426,10.003,149.563
C04646=1122.823,258.248,-71.470,-178.423,10.005,149.563
C04647=1122.818,258.497,-71.499,-178.420,10.008,149.562
C04648=1122.814,258.745,-71.528,-178.416,10.012,149.562
C04649=1122.810,258.993,-71.556,-178.413,10.014,149.562
C04650=1122.805,259.241,-71.586,-178.410,10.017,149.562
C04651=1122.801,259.490,-71.614,-178.407,10.020,149.562
C04652=1122.798,259.738,-71.643,-178.404,10.023,149.562
C04653=1122.792,259.986,-71.672,-178.401,10.026,149.562
C04654=1122.788,260.234,-71.701,-178.398,10.029,149.562
C04655=1122.784,260.483,-71.730,-178.395,10.032,149.562
C04656=1122.780,260.731,-71.759,-178.391,10.035,149.562
C04657=1122.776,260.979,-71.788,-178.388,10.038,149.561
C04658=1122.771,261.228,-71.817,-178.385,10.040,149.561
C04659=1122.767,261.476,-71.846,-178.381,10.044,149.561
C04660=1122.763,261.724,-71.875,-178.379,10.047,149.561
C04661=1122.759,261.973,-71.904,-178.375,10.049,149.561
C04662=1122.754,262.220,-71.933,-178.372,10.053,149.561
C04663=1122.750,262.469,-71.962,-178.368,10.055,149.560
C04664=1122.746,262.718,-71.991,-178.365,10.058,149.560
C04665=1122.741,262.966,-72.020,-178.362,10.061,149.560
C04666=1122.737,263.214,-72.050,-178.358,10.064,149.560
C04667=1122.734,263.462,-72.079,-178.354,10.067,149.559
C04668=1122.729,263.710,-72.107,-178.351,10.070,149.559
C04669=1122.724,263.958,-72.136,-178.347,10.073,149.559
C04670=1122.720,264.207,-72.166,-178.344,10.076,149.559
C04671=1122.716,264.455,-72.195,-178.340,10.079,149.559
C04672=1122.712,264.703,-72.225,-178.338,10.081,149.559
C04673=1122.708,264.952,-72.254,-178.335,10.084,149.558
C04674=1122.703,265.200,-72.283,-178.332,10.086,149.558
C04675=1122.698,265.448,-72.312,-178.329,10.089,149.558
C04676=1122.694,265.696,-72.342,-178.327,10.091,149.558
C04677=1122.690,265.945,-72.371,-178.324,10.094,149.558
C04678=1122.686,266.193,-72.400,-178.322,10.096,149.558
C04679=1122.682,266.406,-72.426,-178.320,10.098,149.558
C04680=1122.679,266.620,-72.451,-178.318,10.100,149.558
C04681=1122.675,266.833,-72.476,-178.315,10.102,149.558
C04682=1122.672,267.046,-72.501,-178.313,10.104,149.558
C04683=1122.668,267.260,-72.526,-178.311,10.106,149.557
C04684=1122.665,267.473,-72.552,-178.308,10.109,149.558
C04685=1122.661,267.685,-72.577,-178.306,10.111,149.557
C04686=1122.657,267.899,-72.602,-178.304,10.113,149.557
C04687=1122.653,268.147,-72.632,-178.301,10.115,149.557
C04688=1122.649,268.395,-72.661,-178.298,10.118,149.557
C04689=1122.644,268.644,-72.691,-178.295,10.120,149.557
C04690=1122.640,268.892,-72.721,-178.293,10.122,149.557
C04691=1122.635,269.140,-72.750,-178.290,10.125,149.557
C04692=1122.631,269.389,-72.780,-178.287,10.128,149.557
C04693=1122.627,269.637,-72.809,-178.284,10.131,149.557
C04694=1122.623,269.885,-72.838,-178.282,10.133,149.556
C04695=1122.619,270.133,-72.869,-178.279,10.135,149.556
C04696=1122.615,270.381,-72.898,-178.276,10.138,149.556
C04697=1122.611,270.629,-72.928,-178.273,10.141,149.556
C04698=1122.606,270.878,-72.957,-178.271,10.143,149.556
C04699=1122.602,271.126,-72.986,-178.268,10.146,149.556
C04700=1122.597,271.375,-73.016,-178.265,10.149,149.556
C04701=1122.594,271.622,-73.047,-178.262,10.151,149.556
C04702=1122.589,271.870,-73.076,-178.259,10.154,149.556
C04703=1122.585,272.119,-73.106,-178.256,10.157,149.556
C04704=1122.581,272.367,-73.135,-178.253,10.160,149.555
C04705=1122.577,272.615,-73.164,-178.251,10.162,149.555
C04706=1122.572,272.863,-73.195,-178.248,10.164,149.555
C04707=1122.568,273.112,-73.225,-178.245,10.167,149.555
C04708=1122.564,273.360,-73.254,-178.242,10.169,149.555
C04709=1122.560,273.607,-73.284,-178.239,10.172,149.555
C04710=1122.556,273.856,-73.314,-178.236,10.175,149.555
C04711=1122.551,274.104,-73.344,-178.233,10.178,149.554
C04712=1122.547,274.352,-73.374,-178.230,10.180,149.554
C04713=1122.543,274.601,-73.404,-178.227,10.183,149.554
C04714=1122.539,274.849,-73.433,-178.224,10.186,149.554
C04715=1122.535,275.097,-73.464,-178.221,10.188,149.554
C04716=1122.530,275.345,-73.493,-178.218,10.191,149.554
C04717=1122.527,275.593,-73.524,-178.215,10.194,149.554
C04718=1122.522,275.841,-73.553,-178.212,10.196,149.553
C04719=1122.518,276.089,-73.584,-178.209,10.199,149.553
C04720=1122.514,276.338,-73.613,-178.206,10.202,149.553
C04721=1122.510,276.585,-73.643,-178.203,10.205,149.553
C04722=1122.505,276.834,-73.674,-178.199,10.207,149.553
C04723=1122.501,277.082,-73.704,-178.196,10.210,149.553
C04724=1122.497,277.330,-73.734,-178.193,10.213,149.553
C04725=1122.493,277.578,-73.764,-178.190,10.216,149.552
C04726=1122.489,277.827,-73.794,-178.187,10.219,149.552
C04727=1122.485,278.074,-73.824,-178.183,10.221,149.552
C04728=1122.480,278.323,-73.854,-178.180,10.224,149.552
C04729=1122.476,278.571,-73.884,-178.177,10.226,149.552
C04730=1122.472,278.819,-73.915,-178.174,10.229,149.552
C04731=1122.468,279.067,-73.945,-178.170,10.232,149.551
C04732=1122.464,279.315,-73.975,-178.167,10.235,149.551
C04733=1122.459,279.564,-74.005,-178.164,10.238,149.551
C04734=1122.456,279.812,-74.035,-178.161,10.240,149.551
C04735=1122.452,280.025,-74.062,-178.158,10.243,149.551
C04736=1122.448,280.238,-74.088,-178.155,10.245,149.550
C04737=1122.444,280.452,-74.114,-178.152,10.247,149.550
C04738=1122.441,280.664,-74.140,-178.149,10.250,149.550
C04739=1122.437,280.878,-74.166,-178.147,10.252,149.550
C04740=1122.433,281.090,-74.192,-178.144,10.254,149.550
C04741=1122.430,281.303,-74.218,-178.140,10.257,149.549
C04742=1122.427,281.518,-74.244,-178.138,10.259,149.549
C04743=1122.422,281.765,-74.275,-178.135,10.261,149.549
C04744=1122.418,282.013,-74.305,-178.132,10.264,149.549
C04745=1122.413,282.261,-74.336,-178.129,10.267,149.549
C04746=1122.410,282.509,-74.366,-178.125,10.269,149.549
C04747=1122.405,282.758,-74.396,-178.122,10.272,149.549
C04748=1122.401,283.006,-74.426,-178.120,10.275,149.548
C04749=1122.397,283.254,-74.457,-178.116,10.277,149.548
C04750=1122.393,283.502,-74.488,-178.113,10.280,149.548
C04751=1122.389,283.750,-74.518,-178.111,10.281,149.548
C04752=1122.384,283.998,-74.549,-178.108,10.284,149.548
C04753=1122.380,284.246,-74.579,-178.104,10.287,149.547
C04754=1122.376,284.494,-74.611,-178.101,10.289,149.547
C04755=1122.372,284.742,-74.641,-178.098,10.292,149.547
C04756=1122.368,284.990,-74.671,-178.095,10.295,149.547
C04757=1122.364,285.238,-74.703,-178.092,10.297,149.547
C04758=1122.359,285.486,-74.733,-178.089,10.300,149.547
C04759=1122.355,285.734,-74.764,-178.086,10.302,149.546
C04760=1122.351,285.983,-74.795,-178.083,10.305,149.546
C04761=1122.347,286.231,-74.825,-178.080,10.307,149.546
C04762=1122.343,286.478,-74.856,-178.077,10.310,149.546
C04763=1122.339,286.727,-74.887,-178.074,10.312,149.546
C04764=1122.334,286.975,-74.917,-178.071,10.315,149.546
C04765=1122.330,287.223,-74.948,-178.068,10.317,149.545
C04766=1122.326,287.471,-74.979,-178.065,10.320,149.545
C04767=1122.322,287.719,-75.010,-178.061,10.322,149.545
C04768=1122.318,287.968,-75.041,-178.058,10.325,149.545
C04769=1122.314,288.215,-75.072,-178.055,10.328,149.545
C04770=1122.310,288.463,-75.102,-178.052,10.330,149.544
C04771=1122.306,288.712,-75.133,-178.050,10.332,149.544
C04772=1122.301,288.959,-75.164,-178.047,10.335,149.544
C04773=1122.298,289.208,-75.195,-178.044,10.338,149.544
C04774=1122.293,289.456,-75.225,-178.040,10.340,149.544
C04775=1122.289,289.703,-75.257,-178.037,10.343,149.544
C04776=1122.285,289.952,-75.288,-178.034,10.345,149.543
C04777=1122.280,290.200,-75.319,-178.031,10.348,149.543
C04778=1122.277,290.447,-75.350,-178.028,10.350,149.543
C04779=1122.273,290.695,-75.381,-178.025,10.353,149.543
C04780=1122.269,290.944,-75.412,-178.021,10.356,149.543
C04781=1122.264,291.192,-75.443,-178.019,10.358,149.543
C04782=1122.260,291.439,-75.474,-178.016,10.360,149.542
C04783=1122.256,291.688,-75.505,-178.013,10.363,149.542
C04784=1122.251,291.936,-75.536,-178.010,10.365,149.542
C04785=1122.248,292.184,-75.567,-178.007,10.368,149.542
C04786=1122.243,292.432,-75.598,-178.004,10.371,149.542
C04787=1122.240,292.680,-75.630,-178.000,10.373,149.541
C04788=1122.235,292.928,-75.661,-177.997,10.376,149.541
C04789=1122.231,293.176,-75.692,-177.994,10.378,149.541
C04790=1122.227,293.424,-75.723,-177.991,10.381,149.541
C04791=1122.223,293.637,-75.750,-177.989,10.383,149.541
C04792=1122.220,293.850,-75.777,-177.986,10.385,149.541
C04793=1122.216,294.063,-75.803,-177.983,10.387,149.541
C04794=1122.213,294.276,-75.831,-177.981,10.389,149.540
C04795=1122.209,294.489,-75.857,-177.979,10.391,149.540
C04796=1122.206,294.702,-75.885,-177.975,10.394,149.540
C04797=1122.202,294.915,-75.911,-177.973,10.396,149.540
C04798=1122.199,295.128,-75.939,-177.971,10.398,149.540
C04799=1122.195,295.377,-75.970,-177.967,10.400,149.540
C04800=1122.190,295.624,-76.001,-177.964,10.403,149.539
C04801=1122.186,295.873,-76.032,-177.961,10.405,149.539
C04802=1122.182,296.120,-76.064,-177.958,10.408,149.539
C04803=1122.178,296.368,-76.096,-177.955,10.411,149.539
C04804=1122.174,296.617,-76.127,-177.952,10.413,149.539
C04805=1122.170,296.864,-76.158,-177.948,10.416,149.538
C04806=1122.166,297.113,-76.189,-177.946,10.419,149.538
C04807=1122.162,297.360,-76.221,-177.942,10.421,149.538
C04808=1122.158,297.608,-76.253,-177.940,10.423,149.538
C04809=1122.154,297.855,-76.284,-177.937,10.425,149.538
C04810=1122.150,298.104,-76.315,-177.934,10.428,149.538
C04811=1122.145,298.352,-76.348,-177.930,10.431,149.537
C04812=1122.141,298.600,-76.379,-177.927,10.433,149.537
C04813=1122.137,298.848,-76.410,-177.924,10.436,149.537
C04814=1122.132,299.096,-76.442,-177.921,10.439,149.537
C04815=1122.129,299.344,-76.474,-177.918,10.441,149.537
C04816=1122.125,299.592,-76.506,-177.915,10.444,149.537
C04817=1122.121,299.839,-76.537,-177.911,10.446,149.536
C04818=1122.116,300.088,-76.569,-177.909,10.449,149.536
C04819=1122.112,300.336,-76.601,-177.906,10.451,149.536
C04820=1122.108,300.583,-76.632,-177.903,10.453,149.536
C04821=1122.104,300.831,-76.664,-177.900,10.456,149.536
C04822=1122.101,301.079,-76.696,-177.897,10.459,149.536
C04823=1122.096,301.321,-76.727,-177.893,10.461,149.535
C04824=1122.092,301.563,-76.758,-177.890,10.464,149.535
C04825=1122.088,301.806,-76.789,-177.887,10.466,149.535
C04826=1122.084,302.048,-76.820,-177.884,10.469,149.535
C04827=1122.080,302.291,-76.851,-177.881,10.471,149.535
C04828=1122.076,302.533,-76.882,-177.879,10.473,149.534
C04829=1122.072,302.775,-76.914,-177.875,10.476,149.534
C04830=1122.068,303.017,-76.945,-177.872,10.479,149.534
C04831=1122.064,303.265,-76.977,-177.869,10.481,149.534
C04832=1122.059,303.513,-77.009,-177.866,10.484,149.534
C04833=1122.055,303.761,-77.040,-177.863,10.486,149.533
C04834=1122.052,304.009,-77.072,-177.860,10.488,149.533
C04835=1122.047,304.257,-77.105,-177.857,10.491,149.533
C04836=1122.043,304.505,-77.136,-177.854,10.493,149.533
C04837=1122.039,304.753,-77.168,-177.851,10.496,149.533
C04838=1122.035,305.001,-77.201,-177.848,10.499,149.533
C04839=1122.031,305.249,-77.232,-177.844,10.501,149.532
C04840=1122.026,305.497,-77.264,-177.842,10.504,149.532
C04841=1122.022,305.745,-77.296,-177.838,10.506,149.532
C04842=1122.019,305.992,-77.329,-177.835,10.509,149.532
C04843=1122.015,306.241,-77.361,-177.832,10.512,149.532
C04844=1122.010,306.488,-77.393,-177.829,10.514,149.532
C04845=1122.007,306.736,-77.425,-177.826,10.517,149.531
C04846=1122.002,306.984,-77.457,-177.823,10.518,149.531
C04847=1121.999,307.203,-77.485,-177.820,10.521,149.531
C04848=1121.995,307.421,-77.513,-177.818,10.523,149.531
C04849=1121.991,307.639,-77.543,-177.814,10.526,149.531
C04850=1121.988,307.858,-77.571,-177.812,10.528,149.531
C04851=1121.984,308.077,-77.600,-177.809,10.530,149.531
C04852=1121.981,308.295,-77.628,-177.807,10.532,149.530
C04853=1121.977,308.513,-77.656,-177.804,10.535,149.530
C04854=1121.974,308.732,-77.684,-177.801,10.536,149.530
C04855=1121.969,308.980,-77.717,-177.798,10.539,149.530
C04856=1121.966,309.228,-77.749,-177.795,10.542,149.530
C04857=1121.961,309.476,-77.782,-177.792,10.544,149.529
C04858=1121.958,309.724,-77.813,-177.788,10.547,149.529
C04859=1121.953,309.971,-77.846,-177.785,10.550,149.529
C04860=1121.949,310.219,-77.878,-177.782,10.552,149.529
C04861=1121.945,310.467,-77.911,-177.779,10.554,149.529
C04862=1121.941,310.715,-77.944,-177.776,10.556,149.529
C04863=1121.937,310.963,-77.976,-177.773,10.559,149.528
C04864=1121.933,311.211,-78.009,-177.770,10.562,149.528
C04865=1121.929,311.459,-78.040,-177.767,10.564,149.528
C04866=1121.925,311.707,-78.074,-177.764,10.567,149.528
C04867=1121.921,311.954,-78.105,-177.761,10.569,149.528
C04868=1121.916,312.202,-78.138,-177.757,10.572,149.527
C04869=1121.912,312.450,-78.171,-177.754,10.575,149.527
C04870=1121.909,312.698,-78.203,-177.751,10.577,149.527
C04871=1121.904,312.945,-78.236,-177.748,10.580,149.527
C04872=1121.901,313.193,-78.268,-177.745,10.582,149.527
C04873=1121.897,313.441,-78.301,-177.742,10.585,149.527
C04874=1121.892,313.690,-78.334,-177.739,10.587,149.526
C04875=1121.889,313.937,-78.366,-177.736,10.589,149.526
C04876=1121.884,314.185,-78.399,-177.733,10.592,149.526
C04877=1121.880,314.433,-78.432,-177.730,10.594,149.526
C04878=1121.877,314.680,-78.465,-177.727,10.597,149.526
C04879=1121.872,314.929,-78.497,-177.723,10.599,149.525
C04880=1121.868,315.177,-78.530,-177.720,10.602,149.525
C04881=1121.864,315.424,-78.563,-177.717,10.605,149.525
C04882=1121.861,315.672,-78.596,-177.714,10.607,149.525
C04883=1121.856,315.920,-78.628,-177.711,10.610,149.525
C04884=1121.852,316.168,-78.661,-177.708,10.612,149.525
C04885=1121.849,316.415,-78.694,-177.704,10.615,149.524
C04886=1121.844,316.664,-78.726,-177.701,10.618,149.524
C04887=1121.840,316.911,-78.760,-177.698,10.620,149.524
C04888=1121.836,317.159,-78.793,-177.695,10.622,149.524
C04889=1121.832,317.406,-78.825,-177.692,10.624,149.524
C04890=1121.828,317.654,-78.858,-177.689,10.627,149.523
C04891=1121.824,317.902,-78.892,-177.686,10.630,149.523
C04892=1121.820,318.150,-78.924,-177.683,10.632,149.523
C04893=1121.816,318.398,-78.957,-177.679,10.635,149.523
C04894=1121.812,318.645,-78.990,-177.676,10.637,149.523
C04895=1121.808,318.893,-79.023,-177.673,10.640,149.522
C04896=1121.804,319.141,-79.056,-177.670,10.643,149.522
C04897=1121.800,319.389,-79.089,-177.667,10.645,149.522
C04898=1121.796,319.636,-79.122,-177.664,10.647,149.522
C04899=1121.792,319.884,-79.156,-177.661,10.650,149.522
C04900=1121.787,320.132,-79.189,-177.657,10.653,149.522
C04901=1121.784,320.379,-79.221,-177.654,10.655,149.521
C04902=1121.780,320.627,-79.254,-177.652,10.657,149.521
C04903=1121.776,320.840,-79.283,-177.648,10.660,149.521
C04904=1121.773,321.053,-79.312,-177.646,10.662,149.521
C04905=1121.770,321.266,-79.340,-177.643,10.664,149.521
C04906=1121.766,321.479,-79.369,-177.640,10.666,149.521
C04907=1121.763,321.691,-79.397,-177.638,10.668,149.520
C04908=1121.759,321.903,-79.425,-177.635,10.670,149.520
C04909=1121.756,322.116,-79.454,-177.633,10.672,149.520
C04910=1121.753,322.330,-79.482,-177.630,10.674,149.520
C04911=1121.749,322.577,-79.515,-177.627,10.677,149.520
C04912=1121.745,322.824,-79.549,-177.624,10.679,149.519
C04913=1121.741,323.072,-79.582,-177.620,10.682,149.519
C04914=1121.737,323.321,-79.616,-177.617,10.685,149.519
C04915=1121.733,323.568,-79.649,-177.614,10.687,149.519
C04916=1121.729,323.816,-79.682,-177.611,10.689,149.519
C04917=1121.725,324.064,-79.715,-177.608,10.692,149.519
C04918=1121.721,324.311,-79.749,-177.604,10.695,149.518
C04919=1121.717,324.559,-79.782,-177.601,10.697,149.518
C04920=1121.713,324.807,-79.816,-177.598,10.700,149.518
C04921=1121.709,325.055,-79.849,-177.595,10.702,149.518
C04922=1121.704,325.302,-79.883,-177.592,10.705,149.518
C04923=1121.700,325.550,-79.916,-177.589,10.708,149.517
C04924=1121.696,325.798,-79.950,-177.586,10.709,149.517
C04925=1121.692,326.045,-79.983,-177.583,10.712,149.517
C04926=1121.689,326.293,-80.017,-177.580,10.714,149.517
C04927=1121.685,326.541,-80.050,-177.576,10.717,149.517
C04928=1121.681,326.789,-80.083,-177.573,10.719,149.516
C04929=1121.677,327.036,-80.117,-177.570,10.722,149.516
C04930=1121.673,327.284,-80.151,-177.567,10.725,149.516
C04931=1121.669,327.532,-80.185,-177.563,10.727,149.516
C04932=1121.664,327.779,-80.218,-177.561,10.730,149.516
C04933=1121.660,328.027,-80.251,-177.557,10.732,149.516
C04934=1121.657,328.275,-80.286,-177.554,10.735,149.515
C04935=1121.653,328.523,-80.319,-177.551,10.737,149.515
C04936=1121.649,328.770,-80.353,-177.548,10.740,149.515
C04937=1121.644,329.018,-80.386,-177.544,10.742,149.515
C04938=1121.641,329.266,-80.421,-177.542,10.744,149.514
C04939=1121.637,329.513,-80.454,-177.539,10.747,149.514
C04940=1121.633,329.760,-80.488,-177.535,10.749,149.514
C04941=1121.629,330.008,-80.521,-177.532,10.752,149.514
C04942=1121.625,330.256,-80.556,-177.529,10.754,149.514
C04943=1121.621,330.504,-80.589,-177.526,10.757,149.514
C04944=1121.617,330.751,-80.623,-177.523,10.759,149.513
C04945=1121.613,330.999,-80.656,-177.520,10.762,149.513
C04946=1121.609,331.247,-80.691,-177.516,10.765,149.513
C04947=1121.605,331.494,-80.725,-177.513,10.767,149.513
C04948=1121.601,331.742,-80.758,-177.510,10.769,149.513
C04949=1121.597,331.990,-80.793,-177.507,10.772,149.513
C04950=1121.593,332.237,-80.826,-177.503,10.775,149.512
C04951=1121.590,332.485,-80.860,-177.500,10.777,149.512
C04952=1121.585,332.733,-80.894,-177.497,10.780,149.512
C04953=1121.581,332.980,-80.928,-177.494,10.782,149.512
C04954=1121.578,333.228,-80.962,-177.491,10.784,149.512
C04955=1121.573,333.476,-80.996,-177.488,10.786,149.511
C04956=1121.569,333.723,-81.030,-177.485,10.789,149.511
C04957=1121.566,333.971,-81.064,-177.482,10.792,149.511
C04958=1121.561,334.219,-81.098,-177.478,10.794,149.511
C04959=1121.558,334.431,-81.128,-177.476,10.796,149.511
C04960=1121.554,334.644,-81.157,-177.473,10.799,149.510
C04961=1121.551,334.856,-81.186,-177.470,10.801,149.510
C04962=1121.548,335.069,-81.215,-177.467,10.803,149.510
C04963=1121.544,335.281,-81.245,-177.465,10.805,149.510
C04964=1121.541,335.494,-81.274,-177.462,10.807,149.510
C04965=1121.538,335.706,-81.303,-177.459,10.810,149.510
C04966=1121.534,335.919,-81.333,-177.457,10.811,149.509
C04967=1121.530,336.167,-81.367,-177.453,10.814,149.509
C04968=1121.526,336.414,-81.401,-177.450,10.816,149.509
C04969=1121.522,336.663,-81.436,-177.447,10.819,149.509
C04970=1121.519,336.910,-81.470,-177.444,10.821,149.509
C04971=1121.515,337.158,-81.504,-177.440,10.824,149.508
C04972=1121.511,337.405,-81.538,-177.437,10.826,149.508
C04973=1121.507,337.652,-81.572,-177.434,10.829,149.508
C04974=1121.503,337.900,-81.607,-177.431,10.832,149.508
C04975=1121.498,338.148,-81.641,-177.427,10.834,149.508
C04976=1121.495,338.395,-81.676,-177.425,10.836,149.507
C04977=1121.491,338.643,-81.710,-177.422,10.838,149.507
C04978=1121.487,338.891,-81.744,-177.419,10.841,149.507
C04979=1121.483,339.138,-81.779,-177.415,10.843,149.507
C04980=1121.480,339.386,-81.813,-177.412,10.846,149.507
C04981=1121.475,339.633,-81.848,-177.409,10.849,149.507
C04982=1121.471,339.881,-81.882,-177.406,10.851,149.506
C04983=1121.467,340.128,-81.917,-177.402,10.853,149.506
C04984=1121.463,340.376,-81.952,-177.399,10.856,149.506
C04985=1121.460,340.623,-81.986,-177.396,10.858,149.506
C04986=1121.456,340.871,-82.020,-177.393,10.861,149.506
C04987=1121.451,341.119,-82.055,-177.389,10.864,149.505
C04988=1121.448,341.366,-82.089,-177.386,10.866,149.505
C04989=1121.443,341.614,-82.124,-177.383,10.869,149.505
C04990=1121.440,341.861,-82.159,-177.380,10.871,149.505
C04991=1121.436,342.109,-82.193,-177.377,10.874,149.505
C04992=1121.432,342.357,-82.228,-177.374,10.875,149.504
C04993=1121.427,342.604,-82.262,-177.371,10.878,149.504
C04994=1121.424,342.851,-82.297,-177.367,10.880,149.504
C04995=1121.420,343.099,-82.332,-177.364,10.883,149.504
C04996=1121.416,343.347,-82.367,-177.361,10.885,149.503
C04997=1121.412,343.594,-82.402,-177.358,10.888,149.503
C04998=1121.408,343.841,-82.436,-177.354,10.891,149.503
C04999=1121.404,344.090,-82.471,-177.351,10.893,149.503
C05000=1121.400,344.336,-82.506,-177.348,10.895,149.503
C05001=1121.396,344.584,-82.541,-177.344,10.898,149.502
C05002=1121.393,344.832,-82.575,-177.342,10.901,149.502
C05003=1121.389,345.079,-82.610,-177.338,10.903,149.502
C05004=1121.385,345.327,-82.645,-177.335,10.906,149.502
C05005=1121.380,345.574,-82.680,-177.332,10.908,149.502
C05006=1121.376,345.822,-82.715,-177.328,10.911,149.501
C05007=1121.373,346.070,-82.749,-177.326,10.912,149.501
C05008=1121.369,346.317,-82.785,-177.323,10.915,149.501
C05009=1121.365,346.565,-82.819,-177.319,10.917,149.501
C05010=1121.361,346.812,-82.855,-177.316,10.920,149.501
C05011=1121.357,347.060,-82.889,-177.313,10.922,149.500
C05012=1121.353,347.307,-82.925,-177.309,10.925,149.500
C05013=1121.350,347.554,-82.960,-177.306,10.927,149.500
C05014=1121.346,347.802,-82.994,-177.303,10.930,149.500
C05015=1121.342,348.015,-83.025,-177.301,10.932,149.500
C05016=1121.339,348.227,-83.055,-177.297,10.934,149.499
C05017=1121.335,348.439,-83.085,-177.295,10.936,149.499
C05018=1121.332,348.652,-83.115,-177.292,10.939,149.499
C05019=1121.329,348.865,-83.146,-177.289,10.940,149.499
C05020=1121.326,349.077,-83.175,-177.287,10.942,149.499
C05021=1121.322,349.289,-83.206,-177.283,10.945,149.499
C05022=1121.319,349.501,-83.236,-177.281,10.947,149.499
C05023=1121.315,349.749,-83.271,-177.277,10.949,149.498
C05024=1121.311,349.997,-83.306,-177.273,10.952,149.498
C05025=1121.307,350.244,-83.342,-177.270,10.955,149.498
C05026=1121.303,350.491,-83.377,-177.267,10.957,149.497
C05027=1121.299,350.739,-83.412,-177.264,10.960,149.497
C05028=1121.296,350.987,-83.447,-177.260,10.962,149.497
C05029=1121.292,351.234,-83.483,-177.256,10.965,149.497
C05030=1121.288,351.481,-83.518,-177.253,10.968,149.497
C05031=1121.284,351.729,-83.553,-177.249,10.970,149.496
C05032=1121.280,351.977,-83.588,-177.246,10.972,149.496
C05033=1121.276,352.224,-83.624,-177.243,10.975,149.496
C05034=1121.272,352.471,-83.659,-177.239,10.978,149.496
C05035=1121.268,352.719,-83.695,-177.235,10.981,149.495
C05036=1121.265,352.966,-83.730,-177.232,10.983,149.495
C05037=1121.261,353.214,-83.766,-177.228,10.985,149.495
C05038=1121.257,353.461,-83.801,-177.225,10.988,149.494
C05039=1121.253,353.708,-83.836,-177.222,10.990,149.494
C05040=1121.249,353.956,-83.871,-177.218,10.993,149.494
C05041=1121.246,354.203,-83.907,-177.214,10.996,149.494
C05042=1121.242,354.451,-83.942,-177.211,10.998,149.494
C05043=1121.237,354.699,-83.978,-177.207,11.000,149.493
C05044=1121.234,354.946,-84.014,-177.204,11.003,149.493
C05045=1121.230,355.193,-84.049,-177.201,11.005,149.493
C05046=1121.226,355.441,-84.085,-177.198,11.008,149.493
C05047=1121.222,355.688,-84.120,-177.194,11.010,149.492
C05048=1121.219,355.936,-84.156,-177.191,11.012,149.492
C05049=1121.215,356.182,-84.192,-177.187,11.016,149.492
C05050=1121.211,356.430,-84.228,-177.183,11.018,149.492
C05051=1121.207,356.678,-84.264,-177.180,11.021,149.491
C05052=1121.203,356.925,-84.299,-177.176,11.023,149.491
C05053=1121.199,357.172,-84.335,-177.173,11.025,149.491
C05054=1121.196,357.420,-84.370,-177.170,11.028,149.490
C05055=1121.191,357.667,-84.406,-177.166,11.030,149.490
C05056=1121.188,357.914,-84.443,-177.163,11.032,149.490
C05057=1121.184,358.162,-84.478,-177.159,11.035,149.490
C05058=1121.180,358.409,-84.514,-177.156,11.037,149.489
C05059=1121.176,358.657,-84.550,-177.153,11.040,149.489
C05060=1121.172,358.905,-84.585,-177.149,11.042,149.489
C05061=1121.169,359.151,-84.622,-177.146,11.044,149.489
C05062=1121.165,359.399,-84.657,-177.142,11.047,149.488
C05063=1121.161,359.647,-84.693,-177.139,11.049,149.488
C05064=1121.158,359.894,-84.730,-177.136,11.052,149.488
C05065=1121.154,360.141,-84.765,-177.132,11.054,149.487
C05066=1121.150,360.389,-84.801,-177.129,11.056,149.487
C05067=1121.146,360.636,-84.837,-177.125,11.059,149.487
C05068=1121.143,360.883,-84.873,-177.122,11.061,149.487
C05069=1121.138,361.131,-84.909,-177.119,11.064,149.487
C05070=1121.135,361.378,-84.945,-177.115,11.066,149.486
C05071=1121.131,361.590,-84.976,-177.112,11.068,149.486
C05072=1121.128,361.803,-85.008,-177.109,11.070,149.486
C05073=1121.125,362.014,-85.038,-177.106,11.073,149.486
C05074=1121.122,362.227,-85.069,-177.104,11.074,149.485
C05075=1121.118,362.439,-85.099,-177.101,11.076,149.485
C05076=1121.115,362.652,-85.131,-177.098,11.079,149.485
C05077=1121.111,362.864,-85.162,-177.095,11.080,149.485
C05078=1121.108,363.077,-85.193,-177.092,11.083,149.485
C05079=1121.105,363.324,-85.229,-177.088,11.085,149.484
C05080=1121.101,363.571,-85.266,-177.085,11.088,149.484
C05081=1121.097,363.818,-85.302,-177.082,11.090,149.484
C05082=1121.094,364.065,-85.338,-177.079,11.092,149.483
C05083=1121.090,364.313,-85.374,-177.075,11.094,149.483
C05084=1121.086,364.560,-85.410,-177.072,11.096,149.483
C05085=1121.082,364.808,-85.446,-177.069,11.099,149.483
C05086=1121.078,365.055,-85.483,-177.065,11.101,149.483
C05087=1121.074,365.302,-85.519,-177.062,11.104,149.482
C05088=1121.071,365.549,-85.555,-177.058,11.106,149.482
C05089=1121.067,365.796,-85.592,-177.055,11.108,149.482
C05090=1121.063,366.043,-85.628,-177.052,11.111,149.482
C05091=1121.059,366.292,-85.665,-177.049,11.113,149.481
C05092=1121.055,366.539,-85.701,-177.045,11.116,149.481
C05093=1121.052,366.786,-85.738,-177.042,11.118,149.481
C05094=1121.048,367.034,-85.774,-177.038,11.121,149.481
C05095=1121.044,367.281,-85.810,-177.036,11.122,149.480
C05096=1121.040,367.528,-85.847,-177.032,11.125,149.480
C05097=1121.037,367.775,-85.883,-177.029,11.127,149.480
C05098=1121.033,368.022,-85.920,-177.026,11.130,149.480
C05099=1121.028,368.270,-85.956,-177.022,11.132,149.479
C05100=1121.026,368.517,-85.993,-177.019,11.135,149.479
C05101=1121.021,368.764,-86.030,-177.016,11.137,149.479
C05102=1121.017,369.012,-86.067,-177.012,11.140,149.479
C05103=1121.014,369.259,-86.103,-177.009,11.142,149.478
C05104=1121.010,369.506,-86.140,-177.005,11.144,149.478
C05105=1121.006,369.753,-86.175,-177.003,11.146,149.478
C05106=1121.003,370.001,-86.213,-177.000,11.148,149.478
C05107=1120.999,370.248,-86.249,-176.996,11.151,149.478
C05108=1120.995,370.495,-86.286,-176.993,11.153,149.477
C05109=1120.991,370.742,-86.322,-176.990,11.156,149.477
C05110=1120.987,370.990,-86.359,-176.986,11.158,149.477
C05111=1120.984,371.237,-86.397,-176.983,11.161,149.477
C05112=1120.980,371.484,-86.433,-176.980,11.163,149.477
C05113=1120.976,371.732,-86.470,-176.977,11.165,149.476
C05114=1120.972,371.979,-86.507,-176.974,11.167,149.476
C05115=1120.968,372.226,-86.543,-176.970,11.170,149.476
C05116=1120.965,372.473,-86.580,-176.967,11.172,149.476
C05117=1120.961,372.721,-86.617,-176.964,11.175,149.475
C05118=1120.957,372.968,-86.654,-176.961,11.177,149.475
C05119=1120.953,373.215,-86.691,-176.958,11.179,149.475
C05120=1120.950,373.462,-86.728,-176.955,11.181,149.475
C05121=1120.946,373.709,-86.765,-176.952,11.184,149.475
C05122=1120.942,373.956,-86.802,-176.948,11.187,149.475
C05123=1120.938,374.204,-86.839,-176.945,11.189,149.474
C05124=1120.935,374.451,-86.876,-176.942,11.192,149.474
C05125=1120.931,374.698,-86.912,-176.938,11.194,149.474
C05126=1120.927,374.946,-86.949,-176.936,11.196,149.474
C05127=1120.925,375.158,-86.981,-176.933,11.199,149.474
C05128=1120.921,375.370,-87.013,-176.930,11.200,149.473
C05129=1120.917,375.582,-87.044,-176.928,11.202,149.473
C05130=1120.915,375.794,-87.076,-176.925,11.205,149.473
C05131=1120.911,376.006,-87.109,-176.922,11.207,149.473
C05132=1120.908,376.219,-87.140,-176.920,11.209,149.473
C05133=1120.905,376.430,-87.172,-176.917,11.210,149.473
C05134=1120.902,376.642,-87.204,-176.914,11.213,149.473
C05135=1120.898,376.889,-87.241,-176.911,11.216,149.472
C05136=1120.894,377.137,-87.278,-176.908,11.217,149.472
C05137=1120.891,377.384,-87.316,-176.905,11.220,149.472
C05138=1120.887,377.631,-87.352,-176.902,11.223,149.472
C05139=1120.883,377.879,-87.390,-176.899,11.225,149.472
C05140=1120.879,378.126,-87.427,-176.895,11.228,149.472
C05141=1120.875,378.373,-87.464,-176.893,11.230,149.472
C05142=1120.872,378.620,-87.502,-176.890,11.232,149.471
C05143=1120.868,378.867,-87.539,-176.887,11.235,149.471
C05144=1120.864,379.114,-87.576,-176.884,11.237,149.471
C05145=1120.861,379.362,-87.614,-176.880,11.240,149.471
C05146=1120.857,379.609,-87.650,-176.877,11.243,149.471
C05147=1120.853,379.856,-87.688,-176.874,11.245,149.471
C05148=1120.849,380.103,-87.725,-176.872,11.247,149.470
C05149=1120.845,380.350,-87.763,-176.869,11.250,149.470
C05150=1120.842,380.598,-87.800,-176.865,11.252,149.470
C05151=1120.838,380.844,-87.838,-176.862,11.255,149.470
C05152=1120.834,381.091,-87.874,-176.859,11.257,149.470
C05153=1120.831,381.339,-87.912,-176.856,11.260,149.470
C05154=1120.827,381.586,-87.949,-176.854,11.262,149.470
C05155=1120.824,381.833,-87.987,-176.851,11.265,149.470
C05156=1120.820,382.080,-88.025,-176.848,11.268,149.470
C05157=1120.816,382.328,-88.062,-176.844,11.270,149.470
C05158=1120.812,382.575,-88.100,-176.842,11.273,149.470
C05159=1120.808,382.821,-88.138,-176.839,11.275,149.469
C05160=1120.805,383.069,-88.175,-176.836,11.277,149.469
C05161=1120.801,383.316,-88.213,-176.833,11.280,149.469
C05162=1120.798,383.563,-88.251,-176.831,11.282,149.469
C05163=1120.793,383.810,-88.287,-176.829,11.284,149.469
C05164=1120.790,384.057,-88.325,-176.826,11.286,149.469
C05165=1120.787,384.304,-88.363,-176.824,11.289,149.469
C05166=1120.782,384.552,-88.401,-176.822,11.291,149.469
C05167=1120.778,384.799,-88.438,-176.820,11.293,149.469
C05168=1120.775,385.046,-88.476,-176.818,11.295,149.470
C05169=1120.772,385.293,-88.514,-176.816,11.298,149.469
C05170=1120.768,385.540,-88.551,-176.814,11.300,149.470
C05171=1120.764,385.787,-88.589,-176.812,11.302,149.470
C05172=1120.760,386.035,-88.627,-176.810,11.304,149.470
C05173=1120.757,386.281,-88.665,-176.808,11.307,149.470
C05174=1120.753,386.528,-88.703,-176.806,11.309,149.470
C05175=1120.749,386.776,-88.739,-176.804,11.311,149.470
C05176=1120.746,387.023,-88.777,-176.803,11.314,149.470
C05177=1120.742,387.270,-88.816,-176.800,11.316,149.470
C05178=1120.738,387.517,-88.854,-176.798,11.318,149.470
C05179=1120.735,387.764,-88.891,-176.797,11.320,149.470
C05180=1120.731,388.011,-88.929,-176.795,11.323,149.471
C05181=1120.727,388.258,-88.966,-176.793,11.325,149.471
C05182=1120.723,388.506,-89.004,-176.791,11.328,149.471
C05183=1120.721,388.717,-89.037,-176.789,11.330,149.471
C05184=1120.717,388.929,-89.070,-176.788,11.332,149.471
C05185=1120.715,389.141,-89.102,-176.786,11.334,149.471
C05186=1120.711,389.354,-89.134,-176.784,11.336,149.472
C05187=1120.707,389.565,-89.167,-176.784,11.338,149.472
C05188=1120.705,389.777,-89.199,-176.782,11.341,149.472
C05189=1120.701,389.989,-89.232,-176.780,11.343,149.472
C05190=1120.698,390.201,-89.264,-176.779,11.345,149.472
C05191=1120.695,390.449,-89.302,-176.777,11.347,149.472
C05192=1120.691,390.695,-89.340,-176.776,11.350,149.473
C05193=1120.688,390.943,-89.378,-176.773,11.353,149.473
C05194=1120.684,391.190,-89.416,-176.772,11.356,149.473
C05195=1120.680,391.437,-89.454,-176.770,11.358,149.473
C05196=1120.677,391.684,-89.492,-176.768,11.361,149.474
C05197=1120.672,391.931,-89.530,-176.767,11.364,149.474
C05198=1120.669,392.178,-89.569,-176.765,11.367,149.474
C05199=1120.666,392.425,-89.607,-176.763,11.369,149.475
C05200=1120.662,392.672,-89.645,-176.761,11.372,149.475
C05201=1120.658,392.919,-89.683,-176.760,11.375,149.475
C05202=1120.655,393.166,-89.720,-176.758,11.378,149.476
C05203=1120.651,393.413,-89.759,-176.756,11.381,149.476
C05204=1120.647,393.660,-89.797,-176.755,11.384,149.476
C05205=1120.644,393.907,-89.834,-176.753,11.386,149.477
C05206=1120.640,394.155,-89.873,-176.752,11.390,149.477
C05207=1120.636,394.401,-89.911,-176.750,11.393,149.477
C05208=1120.632,394.649,-89.949,-176.749,11.396,149.478
C05209=1120.629,394.895,-89.988,-176.747,11.398,149.478
C05210=1120.625,395.142,-90.025,-176.745,11.402,149.479
C05211=1120.621,395.389,-90.064,-176.744,11.405,149.479
C05212=1120.618,395.637,-90.102,-176.742,11.408,149.479
C05213=1120.614,395.884,-90.140,-176.741,11.411,149.480
C05214=1120.611,396.130,-90.179,-176.740,11.414,149.480
C05215=1120.607,396.378,-90.217,-176.738,11.418,149.481
C05216=1120.603,396.624,-90.255,-176.737,11.421,149.481
C05217=1120.599,396.872,-90.293,-176.735,11.423,149.482
C05218=1120.595,397.119,-90.331,-176.733,11.427,149.482
C05219=1120.593,397.365,-90.369,-176.732,11.430,149.483
C05220=1120.589,397.613,-90.408,-176.731,11.434,149.483
C05221=1120.585,397.860,-90.446,-176.729,11.437,149.484
C05222=1120.581,398.106,-90.485,-176.728,11.441,149.484
C05223=1120.578,398.354,-90.523,-176.727,11.444,149.485
C05224=1120.574,398.601,-90.561,-176.725,11.448,149.485
C05225=1120.570,398.848,-90.599,-176.724,11.451,149.486
C05226=1120.567,399.095,-90.638,-176.722,11.454,149.486
C05227=1120.564,399.342,-90.676,-176.721,11.457,149.487
C05228=1120.559,399.588,-90.715,-176.720,11.462,149.488
C05229=1120.556,399.836,-90.753,-176.719,11.465,149.488
C05230=1120.552,400.083,-90.791,-176.717,11.468,149.489
C05231=1120.549,400.330,-90.830,-176.716,11.472,149.489
C05232=1120.545,400.577,-90.868,-176.714,11.475,149.490
C05233=1120.541,400.824,-90.907,-176.713,11.480,149.491
C05234=1120.538,401.071,-90.945,-176.712,11.483,149.491
C05235=1120.533,401.318,-90.984,-176.711,11.487,149.492
C05236=1120.531,401.564,-91.022,-176.709,11.491,149.493
C05237=1120.527,401.812,-91.061,-176.709,11.494,149.493
C05238=1120.524,402.059,-91.099,-176.707,11.498,149.494
C05239=1120.520,402.271,-91.132,-176.706,11.501,149.495
C05240=1120.517,402.483,-91.165,-176.705,11.504,149.495
C05241=1120.514,402.694,-91.199,-176.704,11.508,149.496
C05242=1120.511,402.906,-91.232,-176.703,11.512,149.496
C05243=1120.507,403.118,-91.265,-176.702,11.515,149.497
C05244=1120.504,403.330,-91.298,-176.701,11.518,149.498
C05245=1120.502,403.542,-91.331,-176.701,11.521,149.498
C05246=1120.499,403.753,-91.364,-176.699,11.525,149.499
C05247=1120.495,404.001,-91.402,-176.699,11.529,149.500
C05248=1120.491,404.248,-91.442,-176.697,11.533,149.501
C05249=1120.487,404.494,-91.480,-176.696,11.537,149.501
C05250=1120.484,404.741,-91.518,-176.695,11.542,149.502
C05251=1120.481,404.988,-91.557,-176.694,11.546,149.503
C05252=1120.477,405.236,-91.596,-176.693,11.549,149.504
C05253=1120.473,405.483,-91.635,-176.692,11.554,149.505
C05254=1120.470,405.728,-91.673,-176.691,11.558,149.505
C05255=1120.466,405.976,-91.712,-176.690,11.562,149.506
C05256=1120.462,406.223,-91.751,-176.689,11.567,149.507
C05257=1120.459,406.470,-91.789,-176.688,11.571,149.508
C05258=1120.455,406.717,-91.828,-176.687,11.576,149.509
C05259=1120.452,406.964,-91.867,-176.686,11.580,149.510
C05260=1120.447,407.211,-91.906,-176.685,11.585,149.511
C05261=1120.444,407.458,-91.944,-176.684,11.589,149.512
C05262=1120.441,407.705,-91.983,-176.684,11.594,149.513
C05263=1120.437,407.952,-92.023,-176.683,11.598,149.514
C05264=1120.434,408.199,-92.061,-176.682,11.603,149.515
C05265=1120.430,408.446,-92.100,-176.681,11.608,149.516
C05266=1120.426,408.692,-92.139,-176.680,11.612,149.517
C05267=1120.422,408.939,-92.178,-176.680,11.617,149.518
C05268=1120.419,409.186,-92.216,-176.679,11.621,149.519
C05269=1120.416,409.433,-92.255,-176.678,11.626,149.520
C05270=1120.412,409.680,-92.294,-176.678,11.631,149.521
C05271=1120.408,409.927,-92.334,-176.676,11.636,149.522
C05272=1120.405,410.174,-92.372,-176.676,11.641,149.523
C05273=1120.402,410.422,-92.411,-176.675,11.646,149.524
C05274=1120.397,410.668,-92.450,-176.675,11.650,149.525
C05275=1120.394,410.915,-92.489,-176.674,11.655,149.527
C05276=1120.390,411.162,-92.528,-176.674,11.660,149.528
C05277=1120.387,411.408,-92.567,-176.673,11.666,149.529
C05278=1120.384,411.655,-92.606,-176.672,11.670,149.530
C05279=1120.380,411.902,-92.645,-176.671,11.675,149.531
C05280=1120.376,412.150,-92.684,-176.671,11.681,149.533
C05281=1120.372,412.397,-92.723,-176.670,11.686,149.534
C05282=1120.369,412.644,-92.763,-176.670,11.691,149.535
C05283=1120.366,412.890,-92.801,-176.669,11.696,149.536
C05284=1120.362,413.137,-92.840,-176.669,11.702,149.537
C05285=1120.358,413.384,-92.879,-176.668,11.707,149.539
C05286=1120.354,413.631,-92.919,-176.668,11.713,149.540
C05287=1120.351,413.878,-92.958,-176.667,11.718,149.541
C05288=1120.349,414.125,-92.997,-176.667,11.723,149.543
C05289=1120.346,414.372,-93.036,-176.666,11.729,149.544
C05290=1120.345,414.619,-93.075,-176.666,11.734,149.545
C05291=1120.344,414.866,-93.113,-176.665,11.740,149.547
C05292=1120.343,415.113,-93.153,-176.666,11.745,149.548
C05293=1120.343,415.360,-93.192,-176.665,11.750,149.549
C05294=1120.344,415.607,-93.229,-176.665,11.756,149.551
C05295=1120.344,415.818,-93.263,-176.664,11.761,149.552
C05296=1120.346,416.030,-93.296,-176.664,11.766,149.553
C05297=1120.347,416.241,-93.329,-176.664,11.770,149.554
C05298=1120.349,416.453,-93.362,-176.664,11.775,149.555
C05299=1120.352,416.664,-93.394,-176.664,11.780,149.557
C05300=1120.355,416.877,-93.427,-176.664,11.785,149.558
C05301=1120.358,417.088,-93.460,-176.663,11.791,149.559
C05302=1120.361,417.299,-93.493,-176.663,11.796,149.561
C05303=1119.942,417.299,-93.556,-176.656,11.800,149.560
C05304=1119.939,417.088,-93.523,-176.656,11.795,149.559
C05305=1119.936,416.875,-93.490,-176.656,11.790,149.557
C05306=1119.933,416.664,-93.457,-176.656,11.785,149.556
C05307=1119.930,416.453,-93.424,-176.657,11.780,149.555
C05308=1119.928,416.241,-93.392,-176.657,11.775,149.554
C05309=1119.927,416.029,-93.358,-176.657,11.770,149.552
C05310=1119.925,415.818,-93.325,-176.657,11.765,149.551
C05311=1119.924,415.606,-93.292,-176.658,11.761,149.550
C05312=1119.923,415.360,-93.253,-176.658,11.754,149.549
C05313=1119.924,415.112,-93.215,-176.658,11.749,149.547
C05314=1119.925,414.866,-93.176,-176.659,11.743,149.546
C05315=1119.926,414.618,-93.137,-176.659,11.738,149.545
C05316=1119.927,414.372,-93.098,-176.660,11.732,149.543
C05317=1119.929,414.124,-93.059,-176.660,11.727,149.542
C05318=1119.932,413.878,-93.021,-176.661,11.721,149.540
C05319=1119.936,413.631,-92.981,-176.661,11.716,149.539
C05320=1119.939,413.384,-92.942,-176.662,11.711,149.538
C05321=1119.943,413.137,-92.903,-176.662,11.705,149.537
C05322=1119.946,412.890,-92.864,-176.662,11.700,149.535
C05323=1119.950,412.643,-92.824,-176.664,11.695,149.534
C05324=1119.953,412.396,-92.786,-176.664,11.690,149.533
C05325=1119.957,412.149,-92.746,-176.665,11.684,149.532
C05326=1119.960,411.902,-92.707,-176.665,11.679,149.531
C05327=1119.964,411.655,-92.668,-176.666,11.674,149.530
C05328=1119.968,411.409,-92.629,-176.667,11.669,149.528
C05329=1119.972,411.162,-92.590,-176.667,11.664,149.527
C05330=1119.974,410.915,-92.551,-176.668,11.659,149.526
C05331=1119.978,410.668,-92.513,-176.669,11.654,149.525
C05332=1119.982,410.421,-92.473,-176.670,11.649,149.524
C05333=1119.986,410.174,-92.434,-176.670,11.644,149.523
C05334=1119.989,409.927,-92.395,-176.671,11.639,149.522
C05335=1119.992,409.680,-92.356,-176.671,11.635,149.521
C05336=1119.996,409.433,-92.317,-176.673,11.629,149.519
C05337=1120.000,409.186,-92.279,-176.674,11.625,149.518
C05338=1120.004,408.939,-92.239,-176.674,11.620,149.517
C05339=1120.007,408.693,-92.201,-176.675,11.615,149.516
C05340=1120.010,408.446,-92.162,-176.676,11.611,149.515
C05341=1120.014,408.199,-92.122,-176.677,11.606,149.514
C05342=1120.018,407.951,-92.084,-176.678,11.602,149.514
C05343=1120.021,407.705,-92.045,-176.678,11.597,149.512
C05344=1120.024,407.458,-92.006,-176.679,11.593,149.511
C05345=1120.029,407.211,-91.967,-176.681,11.587,149.511
C05346=1120.033,406.964,-91.928,-176.682,11.583,149.510
C05347=1120.035,406.717,-91.890,-176.683,11.578,149.509
C05348=1120.039,406.470,-91.851,-176.684,11.574,149.508
C05349=1120.043,406.223,-91.812,-176.684,11.569,149.507
C05350=1120.046,405.976,-91.773,-176.685,11.565,149.506
C05351=1120.050,405.730,-91.734,-176.686,11.562,149.505
C05352=1120.054,405.482,-91.696,-176.687,11.557,149.504
C05353=1120.057,405.235,-91.657,-176.688,11.553,149.503
C05354=1120.061,404.989,-91.618,-176.689,11.549,149.503
C05355=1120.064,404.741,-91.580,-176.690,11.544,149.502
C05356=1120.068,404.495,-91.541,-176.692,11.540,149.501
C05357=1120.072,404.247,-91.503,-176.693,11.536,149.500
C05358=1120.075,404.000,-91.463,-176.694,11.532,149.499
C05359=1120.079,403.753,-91.425,-176.695,11.527,149.499
C05360=1120.082,403.541,-91.392,-176.696,11.524,149.498
C05361=1120.085,403.330,-91.359,-176.697,11.521,149.497
C05362=1120.088,403.118,-91.326,-176.698,11.518,149.497
C05363=1120.091,402.906,-91.292,-176.699,11.514,149.496
C05364=1120.095,402.695,-91.259,-176.700,11.511,149.495
C05365=1120.097,402.483,-91.227,-176.701,11.507,149.495
C05366=1120.100,402.271,-91.194,-176.702,11.504,149.494
C05367=1120.104,402.059,-91.160,-176.703,11.500,149.493
C05368=1120.108,401.812,-91.122,-176.704,11.497,149.493
C05369=1120.110,401.565,-91.083,-176.706,11.493,149.492
C05370=1120.115,401.318,-91.045,-176.707,11.489,149.491
C05371=1120.118,401.071,-91.006,-176.708,11.486,149.491
C05372=1120.122,400.824,-90.968,-176.709,11.482,149.490
C05373=1120.125,400.577,-90.929,-176.711,11.478,149.490
C05374=1120.129,400.330,-90.891,-176.712,11.475,149.489
C05375=1120.133,400.083,-90.852,-176.713,11.471,149.488
C05376=1120.136,399.836,-90.814,-176.715,11.467,149.488
C05377=1120.140,399.589,-90.776,-176.716,11.464,149.487
C05378=1120.143,399.343,-90.737,-176.717,11.460,149.486
C05379=1120.147,399.095,-90.698,-176.718,11.457,149.486
C05380=1120.150,398.848,-90.661,-176.720,11.453,149.485
C05381=1120.155,398.601,-90.622,-176.722,11.449,149.485
C05382=1120.158,398.354,-90.584,-176.723,11.446,149.484
C05383=1120.162,398.107,-90.545,-176.725,11.442,149.484
C05384=1120.165,397.861,-90.507,-176.726,11.439,149.483
C05385=1120.169,397.613,-90.468,-176.727,11.435,149.483
C05386=1120.172,397.366,-90.430,-176.729,11.432,149.482
C05387=1120.177,397.119,-90.392,-176.731,11.429,149.482
C05388=1120.180,396.872,-90.354,-176.732,11.426,149.481
C05389=1120.184,396.625,-90.315,-176.733,11.422,149.481
C05390=1120.188,396.378,-90.277,-176.735,11.419,149.480
C05391=1120.191,396.130,-90.239,-176.737,11.416,149.480
C05392=1120.194,395.884,-90.200,-176.738,11.413,149.480
C05393=1120.198,395.637,-90.163,-176.739,11.410,149.479
C05394=1120.202,395.390,-90.124,-176.741,11.406,149.479
C05395=1120.205,395.142,-90.086,-176.742,11.403,149.478
C05396=1120.210,394.896,-90.048,-176.745,11.400,149.478
C05397=1120.213,394.648,-90.010,-176.746,11.397,149.478
C05398=1120.217,394.401,-89.971,-176.747,11.395,149.477
C05399=1120.220,394.155,-89.933,-176.749,11.391,149.477
C05400=1120.224,393.907,-89.895,-176.751,11.388,149.476
C05401=1120.228,393.661,-89.857,-176.752,11.385,149.476
C05402=1120.231,393.413,-89.819,-176.754,11.382,149.476
C05403=1120.234,393.166,-89.781,-176.756,11.379,149.475
C05404=1120.239,392.919,-89.743,-176.757,11.377,149.475
C05405=1120.242,392.672,-89.705,-176.759,11.374,149.475
C05406=1120.247,392.425,-89.667,-176.761,11.371,149.474
C05407=1120.250,392.178,-89.628,-176.763,11.368,149.474
C05408=1120.253,391.931,-89.590,-176.764,11.365,149.474
C05409=1120.257,391.684,-89.552,-176.766,11.363,149.474
C05410=1120.260,391.437,-89.514,-176.768,11.359,149.473
C05411=1120.264,391.190,-89.477,-176.770,11.357,149.473
C05412=1120.268,390.943,-89.438,-176.772,11.354,149.473
C05413=1120.271,390.696,-89.400,-176.773,11.352,149.473
C05414=1120.275,390.449,-89.363,-176.775,11.349,149.472
C05415=1120.278,390.202,-89.325,-176.777,11.346,149.472
C05416=1120.282,389.989,-89.292,-176.778,11.344,149.472
C05417=1120.285,389.777,-89.260,-176.780,11.342,149.472
C05418=1120.288,389.566,-89.227,-176.782,11.339,149.472
C05419=1120.292,389.354,-89.195,-176.783,11.338,149.471
C05420=1120.295,389.142,-89.163,-176.785,11.335,149.471
C05421=1120.298,388.930,-89.130,-176.787,11.333,149.471
C05422=1120.300,388.718,-89.097,-176.787,11.331,149.471
C05423=1120.304,388.506,-89.065,-176.789,11.329,149.471
C05424=1120.307,388.259,-89.027,-176.791,11.326,149.471
C05425=1120.312,388.012,-88.989,-176.793,11.324,149.470
C05426=1120.315,387.764,-88.951,-176.795,11.322,149.470
C05427=1120.319,387.517,-88.914,-176.797,11.319,149.470
C05428=1120.322,387.270,-88.876,-176.799,11.316,149.470
C05429=1120.326,387.023,-88.838,-176.801,11.314,149.470
C05430=1120.330,386.776,-88.800,-176.803,11.311,149.470
C05431=1120.334,386.529,-88.762,-176.805,11.309,149.470
C05432=1120.337,386.282,-88.724,-176.807,11.307,149.470
C05433=1120.341,386.035,-88.687,-176.809,11.305,149.470
C05434=1120.344,385.788,-88.650,-176.811,11.302,149.469
C05435=1120.349,385.541,-88.611,-176.813,11.300,149.469
C05436=1120.352,385.293,-88.573,-176.815,11.298,149.469
C05437=1120.356,385.047,-88.536,-176.817,11.296,149.469
C05438=1120.359,384.799,-88.499,-176.819,11.294,149.469
C05439=1120.363,384.552,-88.461,-176.821,11.291,149.469
C05440=1120.366,384.305,-88.423,-176.823,11.289,149.469
C05441=1120.371,384.058,-88.386,-176.826,11.287,149.469
C05442=1120.374,383.810,-88.348,-176.827,11.286,149.469
C05443=1120.378,383.564,-88.310,-176.829,11.284,149.469
C05444=1120.381,383.316,-88.272,-176.832,11.281,149.469
C05445=1120.385,383.069,-88.235,-176.835,11.278,149.469
C05446=1120.389,382.823,-88.198,-176.837,11.276,149.469
C05447=1120.392,382.575,-88.160,-176.841,11.273,149.469
C05448=1120.396,382.328,-88.123,-176.843,11.271,149.469
C05449=1120.399,382.081,-88.085,-176.847,11.268,149.470
C05450=1120.404,381.833,-88.048,-176.850,11.265,149.470
C05451=1120.407,381.586,-88.010,-176.853,11.263,149.470
